       // Encoder fault from ZSW2_ENC
       "HMI_DB".Encoders."1BR".EncoderFault :=
       "DB_EncCom_1BR".EncoderFault;

       "HMI_DB".Encoders."1BR".ErrorCode :=
       "DB_EncCom_1BR".EncoderErrorCode;

       // Encoder alarm / warning from ZSW2_ENC
       "HMI_DB".Encoders."1BR".EncoderAlarm :=
       "DB_EncCom_1BR".EncoderAlarm;

       // Encoder sign-of-life is valid
       "HMI_DB".Encoders."1BR".EncoderLifeValid :=
       "DB_EncCom_1BR".EncoderLifeValid;


       // ============================================================
       // Preset status
       // ============================================================

       // Preset procedure is active
       "HMI_DB".Encoders."1BR".PresetBusy :=
       "DB_EncCom_1BR".PresetBusy;

       // Preset was done successfully
       "HMI_DB".Encoders."1BR".PresetDone :=
       "DB_EncCom_1BR".PresetDone;

       // Preset error
       "HMI_DB".Encoders."1BR".PresetError :=
       "DB_EncCom_1BR".PresetError;

       // Preset diagnostic status
       "HMI_DB".Encoders."1BR".PresetStatus :=
       "DB_EncCom_1BR".PresetStatus;


       // ============================================================
       // Telegram 89 diagnostic words
       // ============================================================

       // STW2_ENC: control word from PLC to encoder
       "HMI_DB".Encoders."1BR".STW2_ENC :=
       "DB_EncCom_1BR".PzdOutActual.STW2_ENC;

       // ZSW2_ENC: status word from encoder to PLC
       "HMI_DB".Encoders."1BR".ZSW2_ENC :=
       "DB_EncCom_1BR".PzdInActual.ZSW2_ENC;


       // ============================================================
       // General communication FB status
       // ============================================================

       // General diagnostic word of FB_Enc_Tlg89_Com
       "HMI_DB".Encoders."1BR".Status :=
       "DB_EncCom_1BR".Status;

       // -----------------------------------------------------------------------------
       // Масштабоване положення підйому 1BR.
       // -----------------------------------------------------------------------------

       "HMI_DB".Encoders."1BR".Position_mm :=
       LREAL_TO_REAL(
                     "DB_PosCorrection_1BR".ql_PositionCorrected_mm
       );

       "HMI_DB".Encoders."1BR".PositionRounded_mm :=
       "DB_PosCorrection_1BR".qd_PositionCorrectedRounded_mm;

       "HMI_DB".Encoders."1BR".PositionValid :=
       "DB_EncoderScaling".Enc_1BR.PositionValid;

       //======================================

   END_REGION

   //Енкодер пересування візка
   REGION Enc_3BR
       //*********************************
       //Енкодер пересування візка 3BR
       //*********************************

       // ============================================================
       // Main raw values
       // ============================================================

       // Raw position from encoder G1_XIST2
       "HMI_DB".Encoders."3BR".RawPosition :=
       "DB_EncCom_3BR".AbsolutePositionRaw;

       // Raw velocity from encoder NIST_B
       "HMI_DB".Encoders."3BR".RawVelocity :=
       "DB_EncCom_3BR".VelocityRaw;


       // ============================================================
       // Main encoder status
       // ============================================================

       // Encoder is ready for crane logic
       "HMI_DB".Encoders."3BR".EncoderReady :=
       "DB_EncCom_3BR".EncoderReady;

       // Raw position is valid
       "HMI_DB".Encoders."3BR".PositionDataValid :=
       "DB_EncCom_3BR".PositionDataValid;

       // Raw velocity is valid
       "HMI_DB".Encoders."3BR".VelocityDataValid :=
       "DB_EncCom_3BR".VelocityDataValid;

       // Communication fault or cyclic data fault
       "HMI_DB".Encoders."3BR".CommunicationFault :=
       "DB_EncCom_3BR".CommunicationFault;

       // Encoder fault from ZSW2_ENC
       "HMI_DB".Encoders."3BR".EncoderFault :=
       "DB_EncCom_3BR".EncoderFault;

       "HMI_DB".Encoders."3BR".ErrorCode :=
       "DB_EncCom_3BR".EncoderErrorCode;

       // Encoder alarm / warning from ZSW2_ENC
       "HMI_DB".Encoders."3BR".EncoderAlarm :=
       "DB_EncCom_3BR".EncoderAlarm;

       // Encoder sign-of-life is valid
       "HMI_DB".Encoders."3BR".EncoderLifeValid :=
       "DB_EncCom_3BR".EncoderLifeValid;


       // ============================================================
       // Preset status
       // ============================================================

       // Preset procedure is active
       "HMI_DB".Encoders."3BR".PresetBusy :=
       "DB_EncCom_3BR".PresetBusy;

       // Preset was done successfully
       "HMI_DB".Encoders."3BR".PresetDone :=
       "DB_EncCom_3BR".PresetDone;

       // Preset error
       "HMI_DB".Encoders."3BR".PresetError :=
       "DB_EncCom_3BR".PresetError;

       // Preset diagnostic status
       "HMI_DB".Encoders."3BR".PresetStatus :=
       "DB_EncCom_3BR".PresetStatus;


       // ============================================================
       // Telegram 89 diagnostic words
       // ============================================================

       // STW2_ENC: control word from PLC to encoder
       "HMI_DB".Encoders."3BR".STW2_ENC :=
       "DB_EncCom_3BR".PzdOutActual.STW2_ENC;

       // ZSW2_ENC: status word from encoder to PLC
       "HMI_DB".Encoders."3BR".ZSW2_ENC :=
       "DB_EncCom_3BR".PzdInActual.ZSW2_ENC;


       // ============================================================
       // General communication FB status
       // ============================================================

       // General diagnostic word of FB_Enc_Tlg89_Com
       "HMI_DB".Encoders."3BR".Status :=
       "DB_EncCom_3BR".Status;

       // -----------------------------------------------------------------------------
       // Масштабоване положення підйому 1BR.
       // -----------------------------------------------------------------------------

       "HMI_DB".Encoders."3BR".Position_mm :=
       LREAL_TO_REAL(
                     "DB_PosCorrection_3BR".ql_PositionCorrected_mm
       );

       "HMI_DB".Encoders."3BR".PositionRounded_mm :=
       "DB_PosCorrection_3BR".qd_PositionCorrectedRounded_mm;

       "HMI_DB".Encoders."3BR".PositionValid :=
       "DB_EncoderScaling".Enc_3BR.PositionValid;

       //======================================

   END_REGION

   //Енкодер#1 пересування крана
   REGION Enc_4BR1
       //*********************************
       //Енкодер пересування візка 3BR
       //*********************************

       // ============================================================
       // Main raw values
       // ============================================================

       // Raw position from encoder G1_XIST2
       "HMI_DB".Encoders."4BR1".RawPosition :=
       "DB_EncCom_4BR1".AbsolutePositionRaw;

       // Raw velocity from encoder NIST_B
       "HMI_DB".Encoders."4BR1".RawVelocity :=
       "DB_EncCom_4BR1".VelocityRaw;


       // ============================================================
       // Main encoder status
       // ============================================================

       // Encoder is ready for crane logic
       "HMI_DB".Encoders."4BR1".EncoderReady :=
       "DB_EncCom_4BR1".EncoderReady;

       // Raw position is valid
       "HMI_DB".Encoders."4BR1".PositionDataValid :=
       "DB_EncCom_4BR1".PositionDataValid;

       // Raw velocity is valid
       "HMI_DB".Encoders."4BR1".VelocityDataValid :=
       "DB_EncCom_4BR1".VelocityDataValid;

       // Communication fault or cyclic data fault
       "HMI_DB".Encoders."4BR1".CommunicationFault :=
       "DB_EncCom_4BR1".CommunicationFault;

       // Encoder fault from ZSW2_ENC
       "HMI_DB".Encoders."4BR1".EncoderFault :=
       "DB_EncCom_4BR1".EncoderFault;

       "HMI_DB".Encoders."4BR1".ErrorCode :=
       "DB_EncCom_4BR1".EncoderErrorCode;

       // Encoder alarm / warning from ZSW2_ENC
       "HMI_DB".Encoders."4BR1".EncoderAlarm :=
       "DB_EncCom_4BR1".EncoderAlarm;

       // Encoder sign-of-life is valid
       "HMI_DB".Encoders."4BR1".EncoderLifeValid :=
       "DB_EncCom_4BR1".EncoderLifeValid;


       // ============================================================
       // Preset status
       // ============================================================

       // Preset procedure is active
       "HMI_DB".Encoders."4BR1".PresetBusy :=
       "DB_EncCom_4BR1".PresetBusy;

       // Preset was done successfully
       "HMI_DB".Encoders."4BR1".PresetDone :=
       "DB_EncCom_4BR1".PresetDone;

       // Preset error
       "HMI_DB".Encoders."4BR1".PresetError :=
       "DB_EncCom_4BR1".PresetError;

       // Preset diagnostic status
       "HMI_DB".Encoders."4BR1".PresetStatus :=
       "DB_EncCom_4BR1".PresetStatus;


       // ============================================================
       // Telegram 89 diagnostic words
       // ============================================================

       // STW2_ENC: control word from PLC to encoder
       "HMI_DB".Encoders."4BR1".STW2_ENC :=
       "DB_EncCom_4BR1".PzdOutActual.STW2_ENC;

       // ZSW2_ENC: status word from encoder to PLC
       "HMI_DB".Encoders."4BR1".ZSW2_ENC :=
       "DB_EncCom_4BR1".PzdInActual.ZSW2_ENC;


       // ============================================================
       // General communication FB status
       // ============================================================

       // General diagnostic word of FB_Enc_Tlg89_Com
       "HMI_DB".Encoders."4BR1".Status :=
       "DB_EncCom_4BR1".Status;

       // -----------------------------------------------------------------------------
       // Масштабоване положення підйому 1BR.
       // -----------------------------------------------------------------------------

       "HMI_DB".Encoders."4BR1".Position_mm :=
       LREAL_TO_REAL(
                     "DB_PosCorrection_4BR1".ql_PositionCorrected_mm
       );

       "HMI_DB".Encoders."4BR1".PositionRounded_mm :=
       "DB_PosCorrection_4BR1".qd_PositionCorrectedRounded_mm;

       "HMI_DB".Encoders."4BR1".PositionValid :=
       "DB_EncoderScaling".Enc_4BR1.PositionValid;

       //======================================

   END_REGION

   //Енкодер#2 пересування крана
   REGION Enc_4BR2
       //*********************************
       //Енкодер пересування візка 3BR
       //*********************************

       // ============================================================
       // Main raw values
       // ============================================================

       // Raw position from encoder G1_XIST2
       "HMI_DB".Encoders."4BR2".RawPosition :=
       "DB_EncCom_4BR2".AbsolutePositionRaw;

       // Raw velocity from encoder NIST_B
       "HMI_DB".Encoders."4BR2".RawVelocity :=
       "DB_EncCom_4BR2".VelocityRaw;


       // ============================================================
       // Main encoder status
       // ============================================================

       // Encoder is ready for crane logic
       "HMI_DB".Encoders."4BR2".EncoderReady :=
       "DB_EncCom_4BR2".EncoderReady;

       // Raw position is valid
       "HMI_DB".Encoders."4BR2".PositionDataValid :=
       "DB_EncCom_4BR2".PositionDataValid;

       // Raw velocity is valid
       "HMI_DB".Encoders."4BR2".VelocityDataValid :=
       "DB_EncCom_4BR2".VelocityDataValid;

       // Communication fault or cyclic data fault
       "HMI_DB".Encoders."4BR2".CommunicationFault :=
       "DB_EncCom_4BR2".CommunicationFault;

       // Encoder fault from ZSW2_ENC
       "HMI_DB".Encoders."4BR2".EncoderFault :=
       "DB_EncCom_4BR2".EncoderFault;

       "HMI_DB".Encoders."4BR2".ErrorCode :=
       "DB_EncCom_4BR2".EncoderErrorCode;

       // Encoder alarm / warning from ZSW2_ENC
       "HMI_DB".Encoders."4BR2".EncoderAlarm :=
       "DB_EncCom_4BR2".EncoderAlarm;

       // Encoder sign-of-life is valid
       "HMI_DB".Encoders."4BR2".EncoderLifeValid :=
       "DB_EncCom_4BR2".EncoderLifeValid;


       // ============================================================
       // Preset status
       // ============================================================

       // Preset procedure is active
       "HMI_DB".Encoders."4BR2".PresetBusy :=
       "DB_EncCom_4BR2".PresetBusy;

       // Preset was done successfully
       "HMI_DB".Encoders."4BR2".PresetDone :=
       "DB_EncCom_4BR2".PresetDone;

       // Preset error
       "HMI_DB".Encoders."4BR2".PresetError :=
       "DB_EncCom_4BR2".PresetError;

       // Preset diagnostic status
       "HMI_DB".Encoders."4BR2".PresetStatus :=
       "DB_EncCom_4BR2".PresetStatus;


       // ============================================================
       // Telegram 89 diagnostic words
       // ============================================================

       // STW2_ENC: control word from PLC to encoder
       "HMI_DB".Encoders."4BR2".STW2_ENC :=
       "DB_EncCom_4BR2".PzdOutActual.STW2_ENC;

       // ZSW2_ENC: status word from encoder to PLC
       "HMI_DB".Encoders."4BR2".ZSW2_ENC :=
       "DB_EncCom_4BR2".PzdInActual.ZSW2_ENC;


       // ============================================================
       // General communication FB status
       // ============================================================

       // General diagnostic word of FB_Enc_Tlg89_Com
       "HMI_DB".Encoders."4BR2".Status :=
       "DB_EncCom_4BR2".Status;

       // -----------------------------------------------------------------------------
       // Масштабоване положення підйому 1BR.
       // -----------------------------------------------------------------------------

       "HMI_DB".Encoders."4BR2".Position_mm :=
       LREAL_TO_REAL(
                     "DB_PosCorrection_4BR2".ql_PositionCorrected_mm
       );

       "HMI_DB".Encoders."4BR2".PositionRounded_mm :=
       "DB_PosCorrection_4BR2".qd_PositionCorrectedRounded_mm;

       "HMI_DB".Encoders."4BR2".PositionValid :=
       "DB_EncoderScaling".Enc_4BR2.PositionValid;

       //======================================

   END_REGION
END_FUNCTION

FUNCTION "FC_EncoderScale" : Void   // FC82, LAD
{ S7_Optimized_Access := 'TRUE' }
VERSION : 0.1
   VAR_INPUT
      Enable : Bool;   // Загальний дозвіл роботи функції.
      RawPosition : DInt;   // Поточне сире абсолютне положення енкодера.
      RawPositionValid : Bool;   // TRUE — поточне raw-положення достовірне.
      RawPoint1 : DInt;   // Сире значення енкодера у першій контрольній точці.
      PositionPoint1_mm : LReal;   // Координата першої контрольної точки, мм.
      RawPoint2 : DInt;   // Сире значення енкодера у другій контрольній точці.
      PositionPoint2_mm : LReal;   // Координата другої контрольної точки, мм.
   END_VAR
   VAR_OUTPUT
      Position_mm : LReal;   // Розраховане положення механізму, мм.
      PositionRounded_mm : DInt;   // Положення, округлене до цілого міліметра.
      PositionValid : Bool;   // Розраховане положення достовірне. / Результат достовірний і знаходиться в налаштованому діапазоні.
      CalculationValid : Bool;   // Математичний розрахунок виконано за достовірним raw-сигналом.
      ConfigurationValid : Bool;   // Контрольні точки задані коректно.
      InConfiguredRange : Bool;   // Поточне raw-значення знаходиться між двома контрольними точками масштабування. / Поточне raw-значення знаходиться між RawPoint1 і RawPoint2.
      BelowConfiguredRange : Bool;   // Raw-значення нижче мінімальної контрольної raw-точки.
      AboveConfiguredRange : Bool;   // Raw-значення вище максимальної контрольної raw-точки.
      Scale_mm_per_count : LReal;   // Розрахований коефіцієнт масштабування.
      Status : Word;   // Діагностичне слово функції.
   END_VAR
   VAR_TEMP
      RawSpan : LReal;   // Різниця між двома raw-точками.
      PositionSpan_mm : LReal;   // Різниця координат між двома точками, мм.
      RawDelta : LReal;   // Відхилення поточного raw від першої точки.
      RawMinimum : DInt;   // Менша із двох raw-точок.
      RawMaximum : DInt;   // Більша із двох raw-точок.
      CalculatedPosition_mm : LReal;   // Тимчасовий результат масштабування.
   END_VAR
BEGIN

REGION Network 2 (SCL): Розраховане положення механізму, мм.
   // ============================================================
   // 1. Початкові значення виходів
   // ============================================================

   #Position_mm := 0.0;
   #PositionRounded_mm := DINT#0;

   #PositionValid := FALSE;
   #CalculationValid := FALSE;
   #ConfigurationValid := FALSE;

   #InConfiguredRange := FALSE;
   #BelowConfiguredRange := FALSE;
   #AboveConfiguredRange := FALSE;

   #Scale_mm_per_count := 0.0;
   #Status := W#16#0000;

   #RawSpan := 0.0;
   #PositionSpan_mm := 0.0;
   #RawDelta := 0.0;

   #RawMinimum := DINT#0;
   #RawMaximum := DINT#0;

   #CalculatedPosition_mm := 0.0;


   // ============================================================
   // 2. Перевірка дозволу роботи
   // ============================================================

   IF NOT #Enable THEN

       // Bit 0: функція вимкнена.
       #Status := #Status OR W#16#0001;

       RETURN;

   END_IF;


   // ============================================================
   // 3. Перевірка конфігурації контрольних точок
   // ============================================================

   IF #RawPoint1 = #RawPoint2 THEN

       // Bit 2: однакові raw-точки.
       #Status := #Status OR W#16#0004;

   END_IF;


   IF #PositionPoint1_mm = #PositionPoint2_mm THEN

       // Bit 3: однакові координати контрольних точок.
       #Status := #Status OR W#16#0008;

   END_IF;


   #ConfigurationValid :=
   (#RawPoint1 <> #RawPoint2)
   AND
   (#PositionPoint1_mm <> #PositionPoint2_mm);


   IF NOT #ConfigurationValid THEN
       RETURN;
   END_IF;


   // ============================================================
   // 4. Визначення мінімальної та максимальної raw-точок
   // ============================================================

   IF #RawPoint1 < #RawPoint2 THEN

       #RawMinimum := #RawPoint1;
       #RawMaximum := #RawPoint2;

   ELSE

       #RawMinimum := #RawPoint2;
       #RawMaximum := #RawPoint1;

   END_IF;


   // ============================================================
   // 5. Перевірка знаходження raw у налаштованому діапазоні
   // ============================================================

   #BelowConfiguredRange :=
   #RawPosition < #RawMinimum;

   #AboveConfiguredRange :=
   #RawPosition > #RawMaximum;

   #InConfiguredRange :=
   NOT #BelowConfiguredRange
   AND NOT #AboveConfiguredRange;


   IF NOT #InConfiguredRange THEN

       // Bit 4: raw-положення поза налаштованим діапазоном.
       #Status := #Status OR W#16#0010;

   END_IF;


   IF #BelowConfiguredRange THEN

       // Bit 7: raw нижче налаштованого діапазону.
       #Status := #Status OR W#16#0080;

   END_IF;


   IF #AboveConfiguredRange THEN

       // Bit 8: raw вище налаштованого діапазону.
       #Status := #Status OR W#16#0100;

   END_IF;


   // ============================================================
   // 6. Розрахунок коефіцієнта масштабування
   // ============================================================

   // Перетворення виконується до віднімання,
   // щоб уникнути переповнення типу DINT.
   #RawSpan :=
   DINT_TO_LREAL(#RawPoint2)
   - DINT_TO_LREAL(#RawPoint1);

   #PositionSpan_mm :=
   #PositionPoint2_mm
   - #PositionPoint1_mm;

   #Scale_mm_per_count :=
   #PositionSpan_mm
   / #RawSpan;


   // ============================================================
   // 7. Перевірка достовірності вхідного raw-положення
   // ============================================================

   IF NOT #RawPositionValid THEN

       // Bit 1: вхідне raw-положення недостовірне.
       #Status := #Status OR W#16#0002;

       RETURN;

   END_IF;


   // ============================================================
   // 8. Масштабування raw-положення у міліметри
   // ============================================================

   #RawDelta :=
   DINT_TO_LREAL(#RawPosition)
   - DINT_TO_LREAL(#RawPoint1);

   #CalculatedPosition_mm :=
   #PositionPoint1_mm
   + (#RawDelta * #Scale_mm_per_count);

   #Position_mm :=
   #CalculatedPosition_mm;

   #PositionRounded_mm :=
   LREAL_TO_DINT(#CalculatedPosition_mm);

   #CalculationValid := TRUE;

   // Bit 5: математичний розрахунок виконано.
   #Status := #Status OR W#16#0020;


   // ============================================================
   // 9. Формування остаточної валідності положення
   // ============================================================

   #PositionValid :=
   #ConfigurationValid
   AND #RawPositionValid;

   IF #PositionValid THEN

       // Bit 6: результат придатний для штатного використання.
       #Status := #Status OR W#16#0040;

   END_IF;
END_REGION
END_FUNCTION

FUNCTION "FC_AxisProgramLimits" : Void   // FC83, LAD
{ S7_Optimized_Access := 'TRUE' }
VERSION : 0.1
   VAR_INPUT
      Enable : Bool;   // Загальний дозвіл роботи
      Position_mm : LReal;   // Поточне масштабоване положення
      PositionValid : Bool;   // TRUE = положення достовірне
      ProgStopNegative_mm : LReal;   // Нижня програмна межа
      ProgStopPositive_mm : LReal;   // Верхня програмна межа
   END_VAR
   VAR_OUTPUT
      ProgStopNegative : Bool;   // TRUE = досягнута нижня програмна межа
      ProgStopPositive : Bool;   // TRUE = досягнута верхня програмна межа
      ConfigurationValid : Bool;   // TRUE = межі задані коректно
   END_VAR
BEGIN

REGION Network 2 (SCL): Програмні межі
   #ProgStopNegative := FALSE;
   #ProgStopPositive := FALSE;

   #ConfigurationValid :=
   #ProgStopNegative_mm < #ProgStopPositive_mm;

   IF #Enable
       AND #PositionValid
       AND #ConfigurationValid THEN

       #ProgStopNegative :=
       #Position_mm <= #ProgStopNegative_mm;

       #ProgStopPositive :=
       #Position_mm >= #ProgStopPositive_mm;

   END_IF;
END_REGION
END_FUNCTION

FUNCTION "FC_TrolleyPositionLimits" : Void   // FC84, SCL
{ S7_Optimized_Access := 'TRUE' }
VERSION : 0.1
   VAR_INPUT
      Enable : Bool;   // Загальний дозвіл роботи функції
      Position_mm : LReal;   // Поточне скориговане положення механізму візка, мм
      PositionValid : Bool;   // TRUE = положення енкодера достовірне
      BackBuffer_mm : LReal;   // Крайня механічна позиція / буфер назад
      BackEmergencyLimit_mm : LReal;   // Позиція аварійного апаратного кінцевика назад
      BackEncoderLimit_mm : LReal;   // Програмна межа по енкодеру назад
      BackPreStop_mm : LReal;   // Технологічний передзупин назад
      ForwardPreStop_mm : LReal;   // Технологічний передзупин вперед
      ForwardEncoderLimit_mm : LReal;   // Програмна межа по енкодеру вперед
      ForwardEmergencyLimit_mm : LReal;   // Позиція аварійного апаратного кінцевика вперед
      ForwardBuffer_mm : LReal;   // Крайня механічна позиція / буфер вперед
      VirtualOffset_mm : LReal;   // Віртуальне зміщення системи координат, мм
   END_VAR
   VAR_OUTPUT
      BackBuffer : Bool;   // TRUE = досягнута або перевищена позиція буфера назад
      BackEmergencyLimit : Bool;   // TRUE = досягнута позиція аварійного кінцевика назад
      BackEncoderLimit : Bool;   // TRUE = досягнута програмна межа по енкодеру назад
      BackPreStop : Bool;   // TRUE = візок знаходиться в зоні технологічного передзупину назад
      ForwardPreStop : Bool;   // TRUE = візок знаходиться в зоні технологічного передзупину вперед
      ForwardEncoderLimit : Bool;   // TRUE = досягнута програмна межа по енкодеру вперед
      ForwardEmergencyLimit : Bool;   // TRUE = досягнута позиція аварійного кінцевика вперед
      ForwardBuffer : Bool;   // TRUE = досягнута або перевищена позиція буфера вперед
      ConfigurationValid : Bool;   // TRUE = усі координатні уставки задані у правильній послідовності
   END_VAR
BEGIN
   // ============================================================
   // FC_TrolleyPositionLimits
   // Контроль координатних меж і зон механізму візка
   //
   // Негативний напрямок = назад
   // Позитивний напрямок = вперед
   //
   // Послідовність координат:
   //
   // Назад:
   // Буфер -> Аварійний кінцевик -> Межа по енкодеру -> Передзупин
   //
   // Вперед:
   // Передзупин -> Межа по енкодеру -> Аварійний кінцевик -> Буфер
   // ============================================================


   // ============================================================
   // 1. Початкові значення виходів
   // ============================================================

   #BackBuffer := FALSE;
   #BackEmergencyLimit := FALSE;
   #BackEncoderLimit := FALSE;
   #BackPreStop := FALSE;

   #ForwardPreStop := FALSE;
   #ForwardEncoderLimit := FALSE;
   #ForwardEmergencyLimit := FALSE;
   #ForwardBuffer := FALSE;


   // ============================================================
   // 2. Перевірка конфігурації
   //
   // Усі координатні межі повинні бути задані послідовно
   // від заднього буфера до переднього буфера.
   // ============================================================

   #ConfigurationValid :=
   (#BackBuffer_mm < #BackEmergencyLimit_mm)
   AND (#BackEmergencyLimit_mm < #BackEncoderLimit_mm)
   AND (#BackEncoderLimit_mm < #BackPreStop_mm)
   AND (#BackPreStop_mm < #ForwardPreStop_mm)
   AND (#ForwardPreStop_mm < #ForwardEncoderLimit_mm)
   AND (#ForwardEncoderLimit_mm < #ForwardEmergencyLimit_mm)
   AND (#ForwardEmergencyLimit_mm < #ForwardBuffer_mm);


   // ============================================================
   // 3. Розрахунок координатних меж
   //
   // Контроль виконується тільки за умов:
   // - функція дозволена;
   // - положення енкодера достовірне;
   // - конфігурація координатних меж коректна.
   // ============================================================

   IF #Enable
       AND #PositionValid
       AND #ConfigurationValid
   THEN

       // ========================================================
       // 3.1 Рух назад
       //
       // При русі назад координата візка зменшується.
       // Вихід стає TRUE після досягнення відповідної межі.
       // ========================================================

       // Досягнута зона технологічного передзупину назад.
       #BackPreStop :=
       #Position_mm <= (#BackPreStop_mm + #VirtualOffset_mm);

       // Досягнута програмна межа по енкодеру назад.
       #BackEncoderLimit :=
       #Position_mm <= (#BackEncoderLimit_mm + #VirtualOffset_mm);

       // Досягнута позиція аварійного апаратного кінцевика назад.
       #BackEmergencyLimit :=
       #Position_mm <= (#BackEmergencyLimit_mm + #VirtualOffset_mm);

       // Досягнута крайня механічна позиція / буфер назад.
       #BackBuffer :=
       #Position_mm <= (#BackBuffer_mm + #VirtualOffset_mm);


       // ========================================================
       // 3.2 Рух вперед
       //
       // При русі вперед координата візка збільшується.
       // Вихід стає TRUE після досягнення відповідної межі.
       // ========================================================

       // Досягнута зона технологічного передзупину вперед.
       #ForwardPreStop :=
       #Position_mm >= (#ForwardPreStop_mm + #VirtualOffset_mm);

       // Досягнута програмна межа по енкодеру вперед.
       #ForwardEncoderLimit :=
       #Position_mm >=(#ForwardEncoderLimit_mm + #VirtualOffset_mm);

       // Досягнута позиція аварійного апаратного кінцевика вперед.
       #ForwardEmergencyLimit :=
       #Position_mm >= (#ForwardEmergencyLimit_mm + #VirtualOffset_mm);

       // Досягнута крайня механічна позиція / буфер вперед.
       #ForwardBuffer :=
       #Position_mm >= (#ForwardBuffer_mm + #VirtualOffset_mm);

   END_IF;
END_FUNCTION

FUNCTION "FC_HoistPositionLimits" : Void   // FC85, SCL
{ S7_Optimized_Access := 'TRUE' }
VERSION : 0.1
   VAR_INPUT
      Enable : Bool;   // Загальний дозвіл роботи функції
      Position_mm : LReal;   // Поточне скориговане положення механізму підйому, мм
      PositionValid : Bool;   // TRUE = положення енкодера достовірне
      DownEndPosition_mm : LReal;   // Крайня нижня позиція механізму
      DownEmergencyLimit_mm : LReal;   // Позиція аварійного кінцевика при опусканні
      DownEncoderLimit_mm : LReal;   // Програмна межа по енкодеру при опусканні
      DownPreStop_mm : LReal;   // Технологічний передзупин при опусканні
      UpPreStop_mm : LReal;   // Технологічний передзупин при підйомі
      UpEncoderLimit_mm : LReal;   // Програмна межа по енкодеру при підйомі
      UpEmergencyLimit_mm : LReal;   // Позиція аварійного кінцевика при підйомі
      UpEndPosition_mm : LReal;   // Крайня верхня позиція механізму
      VirtualOffset_mm : LReal;   // Віртуальне зміщення системи координат, мм
   END_VAR
   VAR_OUTPUT
      DownEndPosition : Bool;   // Досягнута крайня нижня позиція
      DownEmergencyLimit : Bool;   // Досягнута позиція аварійного кінцевика при опусканні
      DownEncoderLimit : Bool;   // Досягнута програмна межа по енкодеру при опусканні
      DownPreStop : Bool;   // Активна зона технологічного передзупину при опусканні
      UpPreStop : Bool;   // Активна зона технологічного передзупину при підйомі
      UpEncoderLimit : Bool;   // Досягнута програмна межа по енкодеру при підйомі
      UpEmergencyLimit : Bool;   // Досягнута позиція аварійного кінцевика при підйомі
      UpEndPosition : Bool;   // Досягнута крайня верхня позиція
      ConfigurationValid : Bool;   // TRUE = координатні межі задані коректно
   END_VAR
BEGIN
   // ============================================================
   // FC_HoistPositionLimits
   // Контроль координатних меж механізму підйому
   //
   // Підйом     = позитивний напрямок руху.
   // Опускання  = негативний напрямок руху.
   //
   // При підйомі координата збільшується.
   // При опусканні координата зменшується.
   //
   // Послідовність меж при опусканні:
   // Низ -> Аварійний кінцевик -> Межа по енкодеру -> Передзупин
   //
   // Послідовність меж при підйомі:
   // Передзупин -> Межа по енкодеру -> Аварійний кінцевик -> Верх
   // ============================================================


   // ============================================================
   // 1. Початкові значення виходів
   // ============================================================

   #DownEndPosition := FALSE;
   #DownEmergencyLimit := FALSE;
   #DownEncoderLimit := FALSE;
   #DownPreStop := FALSE;

   #UpPreStop := FALSE;
   #UpEncoderLimit := FALSE;
   #UpEmergencyLimit := FALSE;
   #UpEndPosition := FALSE;


   // ============================================================
   // 2. Перевірка конфігурації
   //
   // Координатні межі повинні послідовно збільшуватись
   // від крайньої нижньої позиції до крайньої верхньої позиції.
   // ============================================================

   #ConfigurationValid :=
   (#DownEndPosition_mm < #DownEmergencyLimit_mm)
   AND (#DownEmergencyLimit_mm < #DownEncoderLimit_mm)
   AND (#DownEncoderLimit_mm < #DownPreStop_mm)
   AND (#DownPreStop_mm < #UpPreStop_mm)
   AND (#UpPreStop_mm < #UpEncoderLimit_mm)
   AND (#UpEncoderLimit_mm < #UpEmergencyLimit_mm)
   AND (#UpEmergencyLimit_mm < #UpEndPosition_mm);


   // ============================================================
   // 3. Розрахунок координатних меж
   //
   // Контроль виконується тільки за умов:
   // - функція дозволена;
   // - положення енкодера достовірне;
   // - конфігурація координатних меж коректна.
   // ============================================================

   IF #Enable
       AND #PositionValid
       AND #ConfigurationValid
   THEN

       // ========================================================
       // 3.1 Опускання
       //
       // Опускання є негативним напрямком руху.
       // При опусканні координата зменшується.
       // ========================================================

       // Досягнута зона технологічного передзупину при опусканні.
       #DownPreStop :=
       #Position_mm <= (#DownPreStop_mm + #VirtualOffset_mm);

       // Досягнута програмна межа по енкодеру при опусканні.
       #DownEncoderLimit :=
       #Position_mm <= (#DownEncoderLimit_mm + #VirtualOffset_mm);

       // Досягнута позиція аварійного апаратного кінцевика
       // при опусканні.
       #DownEmergencyLimit :=
       #Position_mm <= (#DownEmergencyLimit_mm + #VirtualOffset_mm);

       // Досягнута крайня нижня позиція механізму.
       #DownEndPosition :=
       #Position_mm <= (#DownEndPosition_mm + #VirtualOffset_mm);


       // ========================================================
       // 3.2 Підйом
       //
       // Підйом є позитивним напрямком руху.
       // При підйомі координата збільшується.
       // ========================================================

       // Досягнута зона технологічного передзупину при підйомі.
       #UpPreStop :=
       #Position_mm >= (#UpPreStop_mm + #VirtualOffset_mm);

       // Досягнута програмна межа по енкодеру при підйомі.
       #UpEncoderLimit :=
       #Position_mm >= (#UpEncoderLimit_mm + #VirtualOffset_mm);

       // Досягнута позиція аварійного апаратного кінцевика
       // при підйомі.
       #UpEmergencyLimit :=
       #Position_mm >= (#UpEmergencyLimit_mm + #VirtualOffset_mm);

       // Досягнута крайня верхня позиція механізму.
       #UpEndPosition :=
       #Position_mm >= (#UpEndPosition_mm + #VirtualOffset_mm);

   END_IF;
END_FUNCTION

FUNCTION "FC_BridgePositionLimits" : Void   // FC86, SCL
{ S7_Optimized_Access := 'TRUE' }
VERSION : 0.1
   VAR_INPUT
      Enable : Bool;   // Загальний дозвіл роботи функції
      Position_mm : LReal;   // Поточне скориговане положення механізму моста, мм
      PositionValid : Bool;   // TRUE = положення енкодера достовірне
      LeftBuffer_mm : LReal;   // Позиція буфера зліва
      LeftEmergencyLimit_mm : LReal;   // Позиція аварійного кінцевика зліва
      LeftEncoderLimit_mm : LReal;   // Програмна межа по енкодеру зліва
      LeftPreStop_mm : LReal;   // Технологічний передзупин при русі вліво
      LeftZoneLimit_mm : LReal;   // Ліва координатна межа зони
      RightZoneLimit_mm : LReal;   // Права координатна межа зони
      RightPreStop_mm : LReal;   // Технологічний передзупин при русі вправо
      RightEncoderLimit_mm : LReal;   // Програмна межа по енкодеру справа
      RightEmergencyLimit_mm : LReal;   // Позиція аварійного кінцевика справа
      RightBuffer_mm : LReal;   // Позиція буфера справа
      VirtualOffset_mm : LReal;   // Віртуальне зміщення системи координат, мм
   END_VAR
   VAR_OUTPUT
      LeftBuffer : Bool;   // Досягнута позиція буфера зліва
      LeftEmergencyLimit : Bool;   // Досягнута позиція аварійного кінцевика зліва
      LeftEncoderLimit : Bool;   // Досягнута програмна межа по енкодеру зліва
      LeftPreStop : Bool;   // Досягнута технологічна межа при русі вліво
      LeftZoneLimit : Bool;   // Досягнута ліва межа зони
      RightZoneLimit : Bool;   // Досягнута права межа зони
      RightPreStop : Bool;   // Досягнута технологічна межа при русі вправо
      RightEncoderLimit : Bool;   // Досягнута програмна межа по енкодеру справа
      RightEmergencyLimit : Bool;   // Досягнута позиція аварійного кінцевика справа
      RightBuffer : Bool;   // Досягнута позиція буфера справа
      ConfigurationValid : Bool;   // TRUE = координатні межі задані коректно
   END_VAR
BEGIN
   // ============================================================
   // FC_BridgePositionLimits
   // Контроль координатних меж механізму моста крана
   //
   // Вправо = позитивний напрямок руху.
   // Вліво  = негативний напрямок руху.
   //
   // При русі вправо координата збільшується.
   // При русі вліво координата зменшується.
   //
   // Послідовність координат:
   //
   // Вліво:
   // Буфер -> Аварійний кінцевик -> Межа по енкодеру
   // -> Технологічний передзупин -> Ліва межа зони
   //
   // Вправо:
   // Права межа зони -> Технологічний передзупин
   // -> Межа по енкодеру -> Аварійний кінцевик -> Буфер
   // ============================================================


   // ============================================================
   // 1. Початкові значення виходів
   // ============================================================

   #LeftBuffer := FALSE;
   #LeftEmergencyLimit := FALSE;
   #LeftEncoderLimit := FALSE;
   #LeftPreStop := FALSE;
   #LeftZoneLimit := FALSE;

   #RightZoneLimit := FALSE;
   #RightPreStop := FALSE;
   #RightEncoderLimit := FALSE;
   #RightEmergencyLimit := FALSE;
   #RightBuffer := FALSE;


   // ============================================================
   // 2. Перевірка конфігурації
   //
   // Координатні межі повинні послідовно збільшуватись
   // від лівого буфера до правого буфера.
   // ============================================================

   #ConfigurationValid :=
   (#LeftBuffer_mm < #LeftEmergencyLimit_mm)
   AND (#LeftEmergencyLimit_mm < #LeftEncoderLimit_mm)
   AND (#LeftEncoderLimit_mm < #LeftPreStop_mm)
   AND (#LeftPreStop_mm < #LeftZoneLimit_mm)
   AND (#LeftZoneLimit_mm < #RightZoneLimit_mm)
   AND (#RightZoneLimit_mm < #RightPreStop_mm)
   AND (#RightPreStop_mm < #RightEncoderLimit_mm)
   AND (#RightEncoderLimit_mm < #RightEmergencyLimit_mm)
   AND (#RightEmergencyLimit_mm < #RightBuffer_mm);


   // ============================================================
   // 3. Розрахунок координатних меж
   //
   // Контроль виконується тільки за умов:
   // - функція дозволена;
   // - положення енкодера достовірне;
   // - конфігурація координатних меж коректна.
   // ============================================================

   IF #Enable
       AND #PositionValid
       AND #ConfigurationValid
   THEN

       // ========================================================
       // 3.1 Рух вліво
       //
       // Вліво є негативним напрямком руху.
       // При русі вліво координата зменшується.
       // ========================================================

       // Досягнута ліва координатна межа зони.
       #LeftZoneLimit :=
       #Position_mm <= (#LeftZoneLimit_mm + #VirtualOffset_mm);

       // Досягнута зона технологічного передзупину
       // при русі вліво.
       #LeftPreStop :=
       #Position_mm <= (#LeftPreStop_mm + #VirtualOffset_mm);

       // Досягнута програмна межа по енкодеру зліва.
       #LeftEncoderLimit :=
       #Position_mm <= (#LeftEncoderLimit_mm + #VirtualOffset_mm);

       // Досягнута позиція аварійного апаратного кінцевика
       // зліва.
       #LeftEmergencyLimit :=
       #Position_mm <= (#LeftEmergencyLimit_mm + #VirtualOffset_mm);

       // Досягнута позиція буфера зліва.
       #LeftBuffer :=
       #Position_mm <= (#LeftBuffer_mm + #VirtualOffset_mm);


       // ========================================================
       // 3.2 Рух вправо
       //
       // Вправо є позитивним напрямком руху.
       // При русі вправо координата збільшується.
       // ========================================================

       // Досягнута права координатна межа зони.
       #RightZoneLimit :=
       #Position_mm >= (#RightZoneLimit_mm + #VirtualOffset_mm);

       // Досягнута зона технологічного передзупину
       // при русі вправо.
       #RightPreStop :=
       #Position_mm >= (#RightPreStop_mm + #VirtualOffset_mm);

       // Досягнута програмна межа по енкодеру справа.
       #RightEncoderLimit :=
       #Position_mm >= (#RightEncoderLimit_mm + #VirtualOffset_mm);

       // Досягнута позиція аварійного апаратного кінцевика
       // справа.
       #RightEmergencyLimit :=
       #Position_mm >= (#RightEmergencyLimit_mm + #VirtualOffset_mm);

       // Досягнута позиція буфера справа.
       #RightBuffer :=
       #Position_mm >= (#RightBuffer_mm + #VirtualOffset_mm);

   END_IF;
END_FUNCTION

// ===== library types =====

TYPE "AnCfg"
   STRUCT
      VRaw : Int;   // Raw value (from input channel)
      LORaw : Int;   // Raw value LO limit
      HIRaw : Int;   // RAW value HI limit
      Val : Real;   // Output value
      LOEng : Real;   // Engineering (scaled) minimum value
      HIEng : Real;   // Engineering (scaled) maximum value
      FVal : Real;   // Filtered value
      PhyVal : Real;   // Physical value (mA)
      LOSP : Real;   // LO setpoint
      LOLOSP : Real;   // LO-LO setpoint
      HISP : Real;   // HI setpoint
      HIHISP : Real;   // HI-HI setpoint
      Hyst : Real;   // Hysteresis in real units
      SimVal : Real;   // Value for simulation
      LOEn : Bool;   // LO warning enabled
      LOLOEn : Bool;   // LO-LO Alarm enabled
      HIEn : Bool;   // HI warning enabled
      HIHIEn : Bool;   // HI-HI Alarm enabled
      LO : Bool;   // Low level is reached
      LOLO : Bool;   // Low Low level is reached
      HI : Bool;   // High level is reached
      HIHI : Bool;   // High High level is reached
      SML : Bool;   // Output value is simulated
      Reset : Bool;   // Reset
      STS : Int;   // Status
      T_FLTR : Int;   // Filtering time, x0.01 seconds
      Text : WString;   // Tag name
      Chanal : WString;   // Chanal
   END_STRUCT;
END_TYPE

(* ===== HMI "HMI_RT_1" =====
system functions are stored by id; their names below are inferred from use
connection "HMI_Connection_1": ETHERNET, S7_1500_OMS

HMI tags "Default tag table"
   "Tag_ScreenNumber" : UInt, internal
   "xAllwaysFalse" : Bool, internal
   "iStep" : Int, internal

HMI tags "DI"
   "HMI_DB_IO_Tags_InCnf_DigIn_0_0" : DigICfg = PLC HMI_DB.IO_Tags.InCnf.DigIn_0_0, 1 s
   "HMI_DB_IO_Tags_InCnf_DigIn_0_1" : DigICfg = PLC HMI_DB.IO_Tags.InCnf.DigIn_0_1 AT %DB1.DBW0, 1 s
   "HMI_DB_IO_Tags_InCnf_DigIn_0_2" : DigICfg = PLC HMI_DB.IO_Tags.InCnf.DigIn_0_2 AT %DB1.DBW0, 1 s
   "HMI_DB_IO_Tags_InCnf_DigIn_0_3" : DigICfg = PLC HMI_DB.IO_Tags.InCnf.DigIn_0_3 AT %DB1.DBW0, 1 s
   "HMI_DB_IO_Tags_InCnf_DigIn_0_4" : DigICfg = PLC HMI_DB.IO_Tags.InCnf.DigIn_0_4 AT %DB1.DBW0, 1 s
   "HMI_DB_IO_Tags_InCnf_DigIn_0_5" : DigICfg = PLC HMI_DB.IO_Tags.InCnf.DigIn_0_5 AT %DB1.DBW0, 1 s
   "HMI_DB_IO_Tags_InCnf_DigIn_0_6" : DigICfg = PLC HMI_DB.IO_Tags.InCnf.DigIn_0_6 AT %DB1.DBW0, 1 s
   "HMI_DB_IO_Tags_InCnf_DigIn_0_7" : DigICfg = PLC HMI_DB.IO_Tags.InCnf.DigIn_0_7 AT %DB1.DBW0, 1 s
   "HMI_DB_IO_Tags_InCnf_DigIn_1_0" : DigICfg = PLC HMI_DB.IO_Tags.InCnf.DigIn_1_0 AT %DB1.DBW0, 1 s
   "HMI_DB_IO_Tags_InCnf_DigIn_1_1" : DigICfg = PLC HMI_DB.IO_Tags.InCnf.DigIn_1_1 AT %DB1.DBW0, 1 s
   "HMI_DB_IO_Tags_InCnf_DigIn_1_2" : DigICfg = PLC HMI_DB.IO_Tags.InCnf.DigIn_1_2 AT %DB1.DBW0, 1 s
   "HMI_DB_IO_Tags_InCnf_DigIn_1_3" : DigICfg = PLC HMI_DB.IO_Tags.InCnf.DigIn_1_3 AT %DB1.DBW0, 1 s
   "HMI_DB_IO_Tags_InCnf_DigIn_1_4" : DigICfg = PLC HMI_DB.IO_Tags.InCnf.DigIn_1_4 AT %DB1.DBW0, 1 s
   "HMI_DB_IO_Tags_InCnf_DigIn_1_5" : DigICfg = PLC HMI_DB.IO_Tags.InCnf.DigIn_1_5 AT %DB1.DBW0, 1 s
   "HMI_DB_IO_Tags_InCnf_DigIn_1_6" : DigICfg = PLC HMI_DB.IO_Tags.InCnf.DigIn_1_6 AT %DB1.DBW0, 1 s
   "HMI_DB_IO_Tags_InCnf_DigIn_1_7" : DigICfg = PLC HMI_DB.IO_Tags.InCnf.DigIn_1_7 AT %DB1.DBW0, 1 s
   "HMI_DB_IO_Tags_InCnf_DigIn_2_0" : DigICfg = PLC HMI_DB.IO_Tags.InCnf.DigIn_2_0 AT %DB1.DBW0, 1 s
   "HMI_DB_IO_Tags_InCnf_DigIn_2_1" : DigICfg = PLC HMI_DB.IO_Tags.InCnf.DigIn_2_1 AT %DB1.DBW0, 1 s
   "HMI_DB_IO_Tags_InCnf_DigIn_2_2" : DigICfg = PLC HMI_DB.IO_Tags.InCnf.DigIn_2_2 AT %DB1.DBW0, 1 s
   "HMI_DB_IO_Tags_InCnf_DigIn_2_3" : DigICfg = PLC HMI_DB.IO_Tags.InCnf.DigIn_2_3 AT %DB1.DBW0, 1 s
   "HMI_DB_IO_Tags_InCnf_DigIn_2_4" : DigICfg = PLC HMI_DB.IO_Tags.InCnf.DigIn_2_4 AT %DB1.DBW0, 1 s
   "HMI_DB_IO_Tags_InCnf_DigIn_2_5" : DigICfg = PLC HMI_DB.IO_Tags.InCnf.DigIn_2_5 AT %DB1.DBW0, 1 s
   "HMI_DB_IO_Tags_InCnf_DigIn_2_6" : DigICfg = PLC HMI_DB.IO_Tags.InCnf.DigIn_2_6 AT %DB1.DBW0, 1 s
   "HMI_DB_IO_Tags_InCnf_DigIn_2_7" : DigICfg = PLC HMI_DB.IO_Tags.InCnf.DigIn_2_7 AT %DB1.DBW0, 1 s
   "HMI_DB_IO_Tags_InCnf_DigIn_3_0" : DigICfg = PLC HMI_DB.IO_Tags.InCnf.DigIn_3_0 AT %DB1.DBW0, 1 s
   "HMI_DB_IO_Tags_InCnf_DigIn_3_1" : DigICfg = PLC HMI_DB.IO_Tags.InCnf.DigIn_3_1 AT %DB1.DBW0, 1 s
   "HMI_DB_IO_Tags_InCnf_DigIn_3_2" : DigICfg = PLC HMI_DB.IO_Tags.InCnf.DigIn_3_2 AT %DB1.DBW0, 1 s
   "HMI_DB_IO_Tags_InCnf_DigIn_3_3" : DigICfg = PLC HMI_DB.IO_Tags.InCnf.DigIn_3_3 AT %DB1.DBW0, 1 s
   "HMI_DB_IO_Tags_InCnf_DigIn_3_4" : DigICfg = PLC HMI_DB.IO_Tags.InCnf.DigIn_3_4 AT %DB1.DBW0, 1 s
   "HMI_DB_IO_Tags_InCnf_DigIn_3_5" : DigICfg = PLC HMI_DB.IO_Tags.InCnf.DigIn_3_5 AT %DB1.DBW0, 1 s
   "HMI_DB_IO_Tags_InCnf_DigIn_3_6" : DigICfg = PLC HMI_DB.IO_Tags.InCnf.DigIn_3_6 AT %DB1.DBW0, 1 s
   "HMI_DB_IO_Tags_InCnf_DigIn_3_7" : DigICfg = PLC HMI_DB.IO_Tags.InCnf.DigIn_3_7 AT %DB1.DBW0, 1 s
   "HMI_DB_IO_Tags_InCnf_DigIn_4_0" : DigICfg = PLC HMI_DB.IO_Tags.InCnf.DigIn_4_0 AT %DB1.DBW0, 1 s
   "HMI_DB_IO_Tags_InCnf_DigIn_4_1" : DigICfg = PLC HMI_DB.IO_Tags.InCnf.DigIn_4_1 AT %DB1.DBW0, 1 s
   "HMI_DB_IO_Tags_InCnf_DigIn_4_2" : DigICfg = PLC HMI_DB.IO_Tags.InCnf.DigIn_4_2 AT %DB1.DBW0, 1 s
   "HMI_DB_IO_Tags_InCnf_DigIn_4_3" : DigICfg = PLC HMI_DB.IO_Tags.InCnf.DigIn_4_3 AT %DB1.DBW0, 1 s
   "HMI_DB_IO_Tags_InCnf_DigIn_4_4" : DigICfg = PLC HMI_DB.IO_Tags.InCnf.DigIn_4_4 AT %DB1.DBW0, 1 s
   "HMI_DB_IO_Tags_InCnf_DigIn_4_5" : DigICfg = PLC HMI_DB.IO_Tags.InCnf.DigIn_4_5 AT %DB1.DBW0, 1 s
   "HMI_DB_IO_Tags_InCnf_DigIn_4_6" : DigICfg = PLC HMI_DB.IO_Tags.InCnf.DigIn_4_6 AT %DB1.DBW0, 1 s
   "HMI_DB_IO_Tags_InCnf_DigIn_4_7" : DigICfg = PLC HMI_DB.IO_Tags.InCnf.DigIn_4_7 AT %DB1.DBW0, 1 s
   "HMI_DB_IO_Tags_InCnf_DigIn_5_0" : DigICfg = PLC HMI_DB.IO_Tags.InCnf.DigIn_5_0 AT %DB1.DBW0, 1 s
   "HMI_DB_IO_Tags_InCnf_DigIn_5_1" : DigICfg = PLC HMI_DB.IO_Tags.InCnf.DigIn_5_1 AT %DB1.DBW0, 1 s
   "HMI_DB_IO_Tags_InCnf_DigIn_5_2" : DigICfg = PLC HMI_DB.IO_Tags.InCnf.DigIn_5_2 AT %DB1.DBW0, 1 s
   "HMI_DB_IO_Tags_InCnf_DigIn_5_3" : DigICfg = PLC HMI_DB.IO_Tags.InCnf.DigIn_5_3 AT %DB1.DBW0, 1 s
   "HMI_DB_IO_Tags_InCnf_DigIn_5_4" : DigICfg = PLC HMI_DB.IO_Tags.InCnf.DigIn_5_4 AT %DB1.DBW0, 1 s
   "HMI_DB_IO_Tags_InCnf_DigIn_5_5" : DigICfg = PLC HMI_DB.IO_Tags.InCnf.DigIn_5_5 AT %DB1.DBW0, 1 s
   "HMI_DB_IO_Tags_InCnf_DigIn_5_6" : DigICfg = PLC HMI_DB.IO_Tags.InCnf.DigIn_5_6 AT %DB1.DBW0, 1 s
   "HMI_DB_IO_Tags_InCnf_DigIn_5_7" : DigICfg = PLC HMI_DB.IO_Tags.InCnf.DigIn_5_7 AT %DB1.DBW0, 1 s
   "HMI_DB_IO_Tags_InCnf_DigIn_6_0" : DigICfg = PLC HMI_DB.IO_Tags.InCnf.DigIn_6_0 AT %DB1.DBW0, 1 s
   "HMI_DB_IO_Tags_InCnf_DigIn_6_1" : DigICfg = PLC HMI_DB.IO_Tags.InCnf.DigIn_6_1 AT %DB1.DBW0, 1 s
   "HMI_DB_IO_Tags_InCnf_DigIn_6_2" : DigICfg = PLC HMI_DB.IO_Tags.InCnf.DigIn_6_2 AT %DB1.DBW0, 1 s
   "HMI_DB_IO_Tags_InCnf_DigIn_6_3" : DigICfg = PLC HMI_DB.IO_Tags.InCnf.DigIn_6_3 AT %DB1.DBW0, 1 s
   "HMI_DB_IO_Tags_InCnf_DigIn_6_4" : DigICfg = PLC HMI_DB.IO_Tags.InCnf.DigIn_6_4 AT %DB1.DBW0, 1 s
   "HMI_DB_IO_Tags_InCnf_DigIn_6_5" : DigICfg = PLC HMI_DB.IO_Tags.InCnf.DigIn_6_5 AT %DB1.DBW0, 1 s
   "HMI_DB_IO_Tags_InCnf_DigIn_6_6" : DigICfg = PLC HMI_DB.IO_Tags.InCnf.DigIn_6_6 AT %DB1.DBW0, 1 s
   "HMI_DB_IO_Tags_InCnf_DigIn_6_7" : DigICfg = PLC HMI_DB.IO_Tags.InCnf.DigIn_6_7 AT %DB1.DBW0, 1 s
   "HMI_DB_IO_Tags_InCnf_DigIn_7_0" : DigICfg = PLC HMI_DB.IO_Tags.InCnf.DigIn_7_0 AT %DB1.DBW0, 1 s
   "HMI_DB_IO_Tags_InCnf_DigIn_7_1" : DigICfg = PLC HMI_DB.IO_Tags.InCnf.DigIn_7_1 AT %DB1.DBW0, 1 s
   "HMI_DB_IO_Tags_InCnf_DigIn_7_2" : DigICfg = PLC HMI_DB.IO_Tags.InCnf.DigIn_7_2 AT %DB1.DBW0, 1 s
   "HMI_DB_IO_Tags_InCnf_DigIn_7_3" : DigICfg = PLC HMI_DB.IO_Tags.InCnf.DigIn_7_3 AT %DB1.DBW0, 1 s
   "HMI_DB_IO_Tags_InCnf_DigIn_7_4" : DigICfg = PLC HMI_DB.IO_Tags.InCnf.DigIn_7_4 AT %DB1.DBW0, 1 s
   "HMI_DB_IO_Tags_InCnf_DigIn_7_5" : DigICfg = PLC HMI_DB.IO_Tags.InCnf.DigIn_7_5 AT %DB1.DBW0, 1 s
   "HMI_DB_IO_Tags_InCnf_DigIn_7_6" : DigICfg = PLC HMI_DB.IO_Tags.InCnf.DigIn_7_6 AT %DB1.DBW0, 1 s
   "HMI_DB_IO_Tags_InCnf_DigIn_7_7" : DigICfg = PLC HMI_DB.IO_Tags.InCnf.DigIn_7_7 AT %DB1.DBW0, 1 s

HMI tags "Internaltags"
   "iVisibilityA1.2" : Bool, internal
   "iVisibilityA1.3" : Bool, internal
   "iVisibilityDevices" : Int, internal

HMI tags "DO"
   "HMI_DB_IO_Tags_OutCfg_DigOut_0_0" : DigOCfg = PLC HMI_DB.IO_Tags.OutCfg.DigOut_0_0, 1 s
   "HMI_DB_IO_Tags_OutCfg_DigOut_0_1" : DigOCfg = PLC HMI_DB.IO_Tags.OutCfg.DigOut_0_1, 1 s
   "HMI_DB_IO_Tags_OutCfg_DigOut_0_2" : DigOCfg = PLC HMI_DB.IO_Tags.OutCfg.DigOut_0_2, 1 s
   "HMI_DB_IO_Tags_OutCfg_DigOut_0_3" : DigOCfg = PLC HMI_DB.IO_Tags.OutCfg.DigOut_0_3, 1 s
   "HMI_DB_IO_Tags_OutCfg_DigOut_0_4" : DigOCfg = PLC HMI_DB.IO_Tags.OutCfg.DigOut_0_4, 1 s
   "HMI_DB_IO_Tags_OutCfg_DigOut_0_5" : DigOCfg = PLC HMI_DB.IO_Tags.OutCfg.DigOut_0_5, 1 s
   "HMI_DB_IO_Tags_OutCfg_DigOut_0_6" : DigOCfg = PLC HMI_DB.IO_Tags.OutCfg.DigOut_0_6, 1 s
   "HMI_DB_IO_Tags_OutCfg_DigOut_0_7" : DigOCfg = PLC HMI_DB.IO_Tags.OutCfg.DigOut_0_7, 1 s
   "HMI_DB_IO_Tags_OutCfg_DigOut_1_0" : DigOCfg = PLC HMI_DB.IO_Tags.OutCfg.DigOut_1_0, 1 s
   "HMI_DB_IO_Tags_OutCfg_DigOut_1_1" : DigOCfg = PLC HMI_DB.IO_Tags.OutCfg.DigOut_1_1, 1 s
   "HMI_DB_IO_Tags_OutCfg_DigOut_1_2" : DigOCfg = PLC HMI_DB.IO_Tags.OutCfg.DigOut_1_2, 1 s
   "HMI_DB_IO_Tags_OutCfg_DigOut_1_3" : DigOCfg = PLC HMI_DB.IO_Tags.OutCfg.DigOut_1_3, 1 s
   "HMI_DB_IO_Tags_OutCfg_DigOut_1_4" : DigOCfg = PLC HMI_DB.IO_Tags.OutCfg.DigOut_1_4, 1 s
   "HMI_DB_IO_Tags_OutCfg_DigOut_1_5" : DigOCfg = PLC HMI_DB.IO_Tags.OutCfg.DigOut_1_5, 1 s
   "HMI_DB_IO_Tags_OutCfg_DigOut_1_6" : DigOCfg = PLC HMI_DB.IO_Tags.OutCfg.DigOut_1_6, 1 s
   "HMI_DB_IO_Tags_OutCfg_DigOut_1_7" : DigOCfg = PLC HMI_DB.IO_Tags.OutCfg.DigOut_1_7, 1 s

HMI tags "AI"
   "HMI_DB_IO_Tags_InAnCfg_AnIn_0" : AnICfg = PLC HMI_DB.IO_Tags.InAnCfg.AnIn_0, 1 s
   "HMI_DB_IO_Tags_InAnCfg_AnIn_1" : AnICfg = PLC HMI_DB.IO_Tags.InAnCfg.AnIn_1, 1 s
   "HMI_DB_IO_Tags_InAnCfg_AnIn_2" : AnICfg = PLC HMI_DB.IO_Tags.InAnCfg.AnIn_2, 1 s
   "HMI_DB_IO_Tags_InAnCfg_AnIn_3" : AnICfg = PLC HMI_DB.IO_Tags.InAnCfg.AnIn_3, 1 s
   "HMI_DB_IO_Tags_InAnCfg_AnIn_4" : AnICfg = PLC HMI_DB.IO_Tags.InAnCfg.AnIn_4, 1 s
   "HMI_DB_IO_Tags_InAnCfg_AnIn_5" : AnICfg = PLC HMI_DB.IO_Tags.InAnCfg.AnIn_5, 1 s
   "HMI_DB_IO_Tags_InAnCfg_AnIn_6" : AnICfg = PLC HMI_DB.IO_Tags.InAnCfg.AnIn_6, 1 s
   "HMI_DB_IO_Tags_InAnCfg_AnIn_7" : AnICfg = PLC HMI_DB.IO_Tags.InAnCfg.AnIn_7, 1 s

HMI tags "Encoders"
   "HMI_DB_Encoders_1BR" : UDT_HMI_Encoder_View = PLC HMI_DB.Encoders.1BR, 1 s
   "HMI_DB_Encoders_3BR" : UDT_HMI_Encoder_View = PLC HMI_DB.Encoders.3BR AT %DB1.DBW0, 1 s
   "HMI_DB_Encoders_4BR1" : UDT_HMI_Encoder_View = PLC HMI_DB.Encoders.4BR1 AT %DB1.DBW0, 1 s
   "HMI_DB_Encoders_4BR2" : UDT_HMI_Encoder_View = PLC HMI_DB.Encoders.4BR2 AT %DB1.DBW0, 1 s

HMI tags "PSMErrors"
   "HMI_DB_Alarms_Contactor_AlarmWord1" : Word = PLC HMI_DB.Alarms.Contactor.AlarmWord1 AT %DB1.DBW0, 1 s
   "HMI_DB_Alarms_Contactor_AlarmWord2" : Word = PLC HMI_DB.Alarms.Contactor.AlarmWord2 AT %DB1.DBW0, 1 s
   "HMI_DB_Alarms_Contactor_AlarmWord3" : Word = PLC HMI_DB.Alarms.Contactor.AlarmWord3 AT %DB1.DBW0, 1 s
   "HMI_DB_PSM_LC_Alarm" : Bool = PLC HMI_DB.PSM.LC_Alarm AT %DB1.DBW0, 1 s

HMI tags "PSM"
   "HMI_DB_PSM_Line_contactor_On" : Bool = PLC HMI_DB.PSM.Line_contactor_On, 1 s
   "HMI_DB_PSM_Control_contactor_220V_On" : Bool = PLC HMI_DB.PSM.Control_contactor_220V_On, 1 s
   "HMI_DB_PSM_Input_voltage_control_380V_On" : Bool = PLC HMI_DB.PSM.Input_voltage_control_380V_On, 1 s
   "HMI_DB_PSM_Heating_circuit_breaker_220V_On" : Bool = PLC HMI_DB.PSM.Heating_circuit_breaker_220V_On, 1 s
   "HMI_DB_PSM_Brake_protection_On" : Bool = PLC HMI_DB.PSM.Brake_protection_On, 1 s
   "HMI_DB_PSM_Transformer_6T1_380V_On" : Bool = PLC HMI_DB.PSM.Transformer_6T1_380V_On, 1 s
   "HMI_DB_PSM_Transformer_sec_circuit_breaker_6T1_380V_On" : Bool = PLC HMI_DB.PSM.Transformer_sec_circuit_breaker_6T1_380V_On, 1 s
   "HMI_DB_PSM_Power_switch_6KV_380V_On" : Bool = PLC HMI_DB.PSM.Power_switch_6KV_380V_On, 1 s
   "HMI_DB_PSM_ID_Control_circuit_breaker_220V_On" : Bool = PLC HMI_DB.PSM.ID_Control_circuit_breaker_220V_On, 1 s
   "HMI_DB_PSM_ID_ORP_power_circuit_breaker_220V_On" : Bool = PLC HMI_DB.PSM.ID_ORP_power_circuit_breaker_220V_On, 1 s
   "HMI_DB_PSM_ID_Line_contactor_from_remote_control_On" : Bool = PLC HMI_DB.PSM.ID_Line_contactor_from_remote_control_On, 1 s
   "HMI_DB_PSM_Transformer_9T1_380V_On" : Bool = PLC HMI_DB.PSM.Transformer_9T1_380V_On, 1 s
   "HMI_DB_PSM_Repair_lighting_switch_12V_On" : Bool = PLC HMI_DB.PSM.Repair_lighting_switch_12V_On, 1 s
   "HMI_DB_PSM_Cabinet_circuit_breaker_220V_On" : Bool = PLC HMI_DB.PSM.Cabinet_circuit_breaker_220V_On, 1 s
   "HMI_DB_PSM_CMD_Line_contactor_enable_permission" : Bool = PLC HMI_DB.PSM.CMD_Line_contactor_enable_permission, 1 s
   "HMI_DB_PSM_CMD_Line_contactor_Off" : Bool = PLC HMI_DB.PSM.CMD_Line_contactor_Off, 1 s
   "HMI_DB_PSM_HL_Line_contactor_On" : Bool = PLC HMI_DB.Messages.Crane.wMessageWord1, 1 s
   "HMI_DB_PSM_HL_Input_voltage_abnormal" : Bool = PLC HMI_DB.PSM.HL_Input_voltage_abnormal, 1 s
   "HMI_DB_PSM_Zero_Protection" : Bool = PLC HMI_DB.PSM.Zero_Protection AT %DB1.DBX0.0, 1 s
   "Data_base_Profinet_Ok" : Bool = PLC HMI_DB.Diagnostics.Profinet_Ok AT %DB1.DBX0.0, 1 s
   "HMI_DB_PSM_ColumnEnable" : Bool = PLC HMI_DB.PSM.ColumnEnable AT %DB1.DBX0.0, 1 s
   "HMI_DB_FireAlarm_Active" : Bool = PLC HMI_DB.FireAlarm.Active AT %DB1.DBX0.0, 1 s

HMI tags "Sensors"
   "HMI_DB_Sensors_Cabinet_heating_control_SU1" : Bool = PLC HMI_DB.Sensors.Cabinet_heating_control_SU1, 1 s
   "HMI_DB_Sensors_Seismic_sensor" : Bool = PLC HMI_DB.Sensors.Seismic_sensor, 1 s
   "HMI_DB_Sensors_Drum_rotation_control" : Bool = PLC HMI_DB.Sensors.Drum_rotation_control, 1 s
   "HMI_DB_Sensors_CMD_Bell_On" : Bool = PLC HMI_DB.Sensors.CMD_Bell_On, 500 ms

HMI tags "RemoteControl"
   "HMI_DB_Remote_control" : udtRemCtrl = PLC HMI_DB.Remote_control, 1 s
   "HMI_DB_Remote_control_1" : Bool = PLC HMI_DB.Remote_control.Btn_Bell AT %DB1.DBX0.0, 1 s

HMI tags "LiftingMechanism"
   "HMI_DB_Lifting_mechanism_Work_control" : Bool = PLC HMI_DB.Lifting_mechanism.Work_control, 1 s
   "HMI_DB_Lifting_mechanism_Brake_wear_control" : Bool = PLC HMI_DB.Lifting_mechanism.Brake_wear_control, 1 s
   "HMI_DB_Lifting_mechanism_MD_disconnected_from_drive" : Bool = PLC HMI_DB.Lifting_mechanism.MD_disconnected_from_drive, 1 s
   "HMI_DB_Lifting_mechanism_Thermal_protection_braking_resistor" : Bool = PLC HMI_DB.Lifting_mechanism.Thermal_protection_braking_resistor, 1 s
   "HMI_DB_Lifting_mechanism_NSP_Upward_movement" : Bool = PLC HMI_DB.Lifting_mechanism.NSP_Upward_movement, 1 s
   "HMI_DB_Lifting_mechanism_NSP_Downward_movement" : Bool = PLC HMI_DB.Lifting_mechanism.NSP_Downward_movement, 1 s
   "HMI_DB_Lifting_mechanism_WP_Upward_movement" : Bool = PLC HMI_DB.Lifting_mechanism.WP_Upward_movement, 1 s
   "HMI_DB_Lifting_mechanism_WP_Downward_movement" : Bool = PLC HMI_DB.Lifting_mechanism.WP_Downward_movement, 1 s
   "HMI_DB_Lifting_mechanism_Exceeding_rated_load_115%" : Bool = PLC HMI_DB.Lifting_mechanism.Exceeding_rated_load_115%, 1 s
   "HMI_DB_Lifting_mechanism_Loosening_ropes" : Bool = PLC HMI_DB.Lifting_mechanism.Loosening_ropes, 1 s
   "HMI_DB_Lifting_mechanism_Motor_temperature_protection" : Bool = PLC HMI_DB.Lifting_mechanism.Motor_temperature_protection, 1 s
   "HMI_DB_Lifting_mechanism_1YB1_Brake released" : Bool = PLC HMI_DB.Lifting_mechanism."1YB1_Brake released", 1 s
   "HMI_DB_Lifting_mechanism_1YB1_Brake_applied" : Bool = PLC HMI_DB.Lifting_mechanism.1YB1_Brake_applied, 1 s
   "HMI_DB_Lifting_mechanism_1YB1_Thickness_brake_pads_normal" : Bool = PLC HMI_DB.Lifting_mechanism.1YB1_Thickness_brake_pads_normal, 1 s
   "HMI_DB_Lifting_mechanism_1YB2_Brake released" : Bool = PLC HMI_DB.Lifting_mechanism."1YB2_Brake released", 1 s
   "HMI_DB_Lifting_mechanism_1YB2_Brake_applied" : Bool = PLC HMI_DB.Lifting_mechanism.1YB2_Brake_applied, 1 s
   "HMI_DB_Lifting_mechanism_1YB2_WP_MPP_disconnected_from_brake" : Bool = PLC HMI_DB.Lifting_mechanism.1YB2_WP_MPP_disconnected_from_brake, 1 s
   "HMI_DB_Lifting_mechanism_1YB1_Brake_rectifier_protection" : Bool = PLC HMI_DB.Lifting_mechanism.1YB1_Brake_rectifier_protection, 1 s
   "HMI_DB_Lifting_mechanism_1YB2_Brake_rectifier_protection" : Bool = PLC HMI_DB.Lifting_mechanism.1YB2_Brake_rectifier_protection, 1 s
   "HMI_DB_Lifting_mechanism_CMD_Service_brake_On" : Bool = PLC HMI_DB.Lifting_mechanism.CMD_Service_brake_On, 1 s
   "HMI_DB_Lifting_mechanism_CMD_Built-in_brake_On" : Bool = PLC HMI_DB.Lifting_mechanism.CMD_Built-in_brake_On, 1 s
   "HMI_DB_Lifting_mechanism_CMD_Emergency_brake_On" : Bool = PLC HMI_DB.Lifting_mechanism.CMD_Emergency_brake_On, 1 s
   "HMI_DB_Lifting_mechanism_HL_Drive_ready" : Bool = PLC HMI_DB.Lifting_mechanism.HL_Drive_ready, 1 s
   "HMI_DB_Lifting_mechanism_Torque_control" : Real = PLC HMI_DB.Lifting_mechanism.Torque_control, 1 s
   "HMI_DB_Lifting_mechanism_LM_Alarm" : Bool = PLC HMI_DB.Lifting_mechanism.LM_Alarm AT %DB1.DBX0.0, 1 s
   "HMI_DB_Lifting_mechanism_LM_Status" : Word = PLC HMI_DB.Lifting_mechanism.LM_Status AT %DB1.DBX0.0, 1 s
   "HMI_DB_Lifting_mechanism_NSP_Enable_movement" : Bool = PLC HMI_DB.Lifting_mechanism.NSP_Enable_movement AT %DB1.DBX0.0, 1 s
   "HMI_DB_Lifting_mechanism_SecondSpeedUp" : Bool = PLC HMI_DB.Lifting_mechanism.SecondSpeedUp AT %DB1.DBX0.0, 1 s
   "HMI_DB_Lifting_mechanism_SecondSpeedDown" : Bool = PLC HMI_DB.Lifting_mechanism.SecondSpeedDown, 1 s
   "HMI_DB_Lifting_mechanism_FirstSpeedUp" : Bool = PLC HMI_DB.Lifting_mechanism.FirstSpeedUp AT %DB1.DBX0.0, 1 s
   "HMI_DB_Lifting_mechanism_FirstSpeedDown" : Bool = PLC HMI_DB.Lifting_mechanism.FirstSpeedDown AT %DB1.DBX0.0, 1 s
   "HMI_DB_Calibration_Hoist_Active" : Bool = PLC HMI_DB.Calibration.Hoist.Active AT %DB1.DBX0.0, 1 s
   "HMI_DB_Calibration_Hoist_Calibrated" : Bool = PLC HMI_DB.Calibration.Hoist.Calibrated AT %DB1.DBX0.0, 1 s
   "HMI_DB_Calibration_Hoist_Fault" : Bool = PLC HMI_DB.Calibration.Hoist.Fault AT %DB1.DBX0.0, 1 s
   "HMI_DB_Calibration_Hoist_Aborted" : Bool = PLC HMI_DB.Calibration.Hoist.Aborted AT %DB1.DBX0.0, 1 s
   "HMI_DB_Calibration_Hoist_CurrentStep" : UInt = PLC HMI_DB.Calibration.Hoist.CurrentStep AT %DB1.DBX0.0, 1 s
   "HMI_DB_Calibration_Hoist_CompletedSteps" : DWord = PLC HMI_DB.Calibration.Hoist.CompletedSteps AT %DB1.DBX0.0, 1 s
   "HMI_DB_Calibration_Hoist_Reference1K1" : Bool = PLC HMI_DB.Calibration.Hoist.Reference1K1 AT %DB1.DBX0.0, 1 s
   "HMI_DB_Calibration_Hoist_Position_mm" : DInt = PLC HMI_DB.Calibration.Hoist.Position_mm AT %DB1.DBX0.0, 1 s
   "HMI_DB_Calibration_Hoist_DriveVelocity_rpm" : Real = PLC HMI_DB.Calibration.Hoist.DriveVelocity_rpm AT %DB1.DBX0.0, 1 s
   "HMI_DB_Calibration_Hoist_TimerRemaining" : Time = PLC HMI_DB.Calibration.Hoist.TimerRemaining AT %DB1.DBX0.0, 1 s
   "HMI_DB_Calibration_Hoist_Steps_Completed_Step10" : Bool = PLC HMI_DB.Calibration.Hoist.Steps_Completed.Step10 AT %DB1.DBX0.0, 1 s
   "HMI_DB_Calibration_Hoist_Steps_Completed_Step20" : Bool = PLC HMI_DB.Calibration.Hoist.Steps_Completed.Step20 AT %DB1.DBX0.0, 1 s
   "HMI_DB_Calibration_Hoist_Steps_Completed_Step30" : Bool = PLC HMI_DB.Calibration.Hoist.Steps_Completed.Step30 AT %DB1.DBX0.0, 1 s
   "HMI_DB_Calibration_Hoist_Steps_Completed_Step40" : Bool = PLC HMI_DB.Calibration.Hoist.Steps_Completed.Step40 AT %DB1.DBX0.0, 1 s
   "HMI_DB_Calibration_Hoist_Steps_Completed_Step50" : Bool = PLC HMI_DB.Calibration.Hoist.Steps_Completed.Step50 AT %DB1.DBX0.0, 1 s
   "HMI_DB_Calibration_Hoist_Steps_Completed_Step60" : Bool = PLC HMI_DB.Calibration.Hoist.Steps_Completed.Step60 AT %DB1.DBX0.0, 1 s
   "HMI_DB_Calibration_Hoist_Steps_Completed_Step70" : Bool = PLC HMI_DB.Calibration.Hoist.Steps_Completed.Step70 AT %DB1.DBX0.0, 1 s
   "HMI_DB_Calibration_Hoist_Steps_Completed_Step80" : Bool = PLC HMI_DB.Calibration.Hoist.Steps_Completed.Step80 AT %DB1.DBX0.0, 1 s
   "HMI_DB_Calibration_Hoist_Steps_Completed_Step90" : Bool = PLC HMI_DB.Calibration.Hoist.Steps_Completed.Step90 AT %DB1.DBX0.0, 1 s
   "HMI_DB_Calibration_Hoist_Steps_Completed_Step100" : Bool = PLC HMI_DB.Calibration.Hoist.Steps_Completed.Step100 AT %DB1.DBX0.0, 1 s
   "HMI_DB_Calibration_Hoist_Steps_Completed_Step110" : Bool = PLC HMI_DB.Calibration.Hoist.Steps_Completed.Step110 AT %DB1.DBX0.0, 1 s
   "HMI_DB_Calibration_Hoist_Steps_Completed_Step120" : Bool = PLC HMI_DB.Calibration.Hoist.Steps_Completed.Step120 AT %DB1.DBX0.0, 1 s
   "HMI_DB_Calibration_Hoist_Steps_Completed_Step130" : Bool = PLC HMI_DB.Calibration.Hoist.Steps_Completed.Step130 AT %DB1.DBX0.0, 1 s
   "HMI_DB_Calibration_Hoist_Steps_Active_Step10" : Bool = PLC HMI_DB.Calibration.Hoist.Steps_Active.Step10 AT %DB1.DBX0.0, 1 s
   "HMI_DB_Calibration_Hoist_Steps_Active_Step20" : Bool = PLC HMI_DB.Calibration.Hoist.Steps_Active.Step20 AT %DB1.DBX0.0, 1 s
   "HMI_DB_Calibration_Hoist_Steps_Active_Step30" : Bool = PLC HMI_DB.Calibration.Hoist.Steps_Active.Step30 AT %DB1.DBX0.0, 1 s
   "HMI_DB_Calibration_Hoist_Steps_Active_Step40" : Bool = PLC HMI_DB.Calibration.Hoist.Steps_Active.Step40 AT %DB1.DBX0.0, 1 s
   "HMI_DB_Calibration_Hoist_Steps_Active_Step50" : Bool = PLC HMI_DB.Calibration.Hoist.Steps_Active.Step50 AT %DB1.DBX0.0, 1 s
   "HMI_DB_Calibration_Hoist_Steps_Active_Step60" : Bool = PLC HMI_DB.Calibration.Hoist.Steps_Active.Step60 AT %DB1.DBX0.0, 1 s
   "HMI_DB_Calibration_Hoist_Steps_Active_Step70" : Bool = PLC HMI_DB.Calibration.Hoist.Steps_Active.Step70 AT %DB1.DBX0.0, 1 s
   "HMI_DB_Calibration_Hoist_Steps_Active_Step80" : Bool = PLC HMI_DB.Calibration.Hoist.Steps_Active.Step80 AT %DB1.DBX0.0, 1 s
   "HMI_DB_Calibration_Hoist_Steps_Active_Step90" : Bool = PLC HMI_DB.Calibration.Hoist.Steps_Active.Step90 AT %DB1.DBX0.0, 1 s
   "HMI_DB_Calibration_Hoist_Steps_Active_Step100" : Bool = PLC HMI_DB.Calibration.Hoist.Steps_Active.Step100 AT %DB1.DBX0.0, 1 s
   "HMI_DB_Calibration_Hoist_Steps_Active_Step110" : Bool = PLC HMI_DB.Calibration.Hoist.Steps_Active.Step110 AT %DB1.DBX0.0, 1 s
   "HMI_DB_Calibration_Hoist_Steps_Active_Step120" : Bool = PLC HMI_DB.Calibration.Hoist.Steps_Active.Step120 AT %DB1.DBX0.0, 1 s
   "HMI_DB_Calibration_Hoist_Steps_Active_Step130" : Bool = PLC HMI_DB.Calibration.Hoist.Steps_Active.Step130 AT %DB1.DBX0.0, 1 s
   "HMI_DB_Calibration_Hoist_TimerRemaining_Min" : UInt = PLC HMI_DB.Calibration.Hoist.TimerRemaining_Min AT %DB1.DBX0.0, 1 s
   "HMI_DB_Calibration_Hoist_TimerRemaining_Sec" : UInt = PLC HMI_DB.Calibration.Hoist.TimerRemaining_Sec AT %DB1.DBX0.0, 1 s
   "HMI_DB_Calibration_Hoist_Diagnostics_EncoderControlHealthy" : Bool = PLC HMI_DB.Calibration.Hoist.Diagnostics.EncoderControlHealthy AT %DB1.DBX0.0, 1 s
   "HMI_DB_Calibration_Hoist_Diagnostics_StartupDataConsistent" : Bool = PLC HMI_DB.Calibration.Hoist.Diagnostics.StartupDataConsistent AT %DB1.DBX0.0, 1 s
   "HMI_DB_Calibration_Hoist_Diagnostics_NoMovementWithoutCommand" : Bool = PLC HMI_DB.Calibration.Hoist.Diagnostics.NoMovementWithoutCommand AT %DB1.DBX0.0, 1 s
   "HMI_DB_Calibration_Hoist_Diagnostics_NoManualMovementDetected" : Bool = PLC HMI_DB.Calibration.Hoist.Diagnostics.NoManualMovementDetected AT %DB1.DBX0.0, 1 s
   "HMI_DB_Calibration_Hoist_Diagnostics_EncoderUpdatesDuringMotion" : Bool = PLC HMI_DB.Calibration.Hoist.Diagnostics.EncoderUpdatesDuringMotion AT %DB1.DBX0.0, 1 s
   "HMI_DB_Calibration_Hoist_Diagnostics_EncoderReplacementNotDetected" : Bool = PLC HMI_DB.Calibration.Hoist.Diagnostics.EncoderReplacementNotDetected AT %DB1.DBX0.0, 1 s

HMI tags "TrolleyMovementMechanism"
   "HMI_DB_Trolley_movement_mechanism_Engine_temperature_protection" : Bool = PLC HMI_DB.Trolley_movement_mechanism.Engine_temperature_protection, 1 s
   "HMI_DB_Trolley_movement_mechanism_NSP_Forward_movement" : Bool = PLC HMI_DB.Trolley_movement_mechanism.NSP_Forward_movement, 1 s
   "HMI_DB_Trolley_movement_mechanism_WP_Forward_movement" : Bool = PLC HMI_DB.Trolley_movement_mechanism.WP_Forward_movement, 1 s
   "HMI_DB_Trolley_movement_mechanism_NSP_Backward_movement" : Bool = PLC HMI_DB.Trolley_movement_mechanism.NSP_Backward_movement, 1 s
   "HMI_DB_Trolley_movement_mechanism_WP_Backward_movement" : Bool = PLC HMI_DB.Trolley_movement_mechanism.WP_Backward_movement, 1 s
   "HMI_DB_Trolley_movement_mechanism_MD_disconnected_from_drive" : Bool = PLC HMI_DB.Trolley_movement_mechanism.MD_disconnected_from_drive, 1 s
   "HMI_DB_Trolley_movement_mechanism_Motor_temperature_protection" : Bool = PLC HMI_DB.Trolley_movement_mechanism.Motor_temperature_protection, 1 s
   "HMI_DB_Trolley_movement_mechanism_CMD_Service_brake_On" : Bool = PLC HMI_DB.Trolley_movement_mechanism.CMD_Service_brake_On, 1 s
   "HMI_DB_Trolley_movement_mechanism_HL_Drive_ready" : Bool = PLC HMI_DB.Trolley_movement_mechanism.HL_Drive_ready, 1 s
   "HMI_DB_Trolley_movement_mechanism_TM_Status" : Word = PLC HMI_DB.Trolley_movement_mechanism.TM_Status AT %DB1.DBX0.0, 1 s
   "HMI_DB_Trolley_movement_mechanism_NSP_Enable_movement" : Bool = PLC HMI_DB.Trolley_movement_mechanism.NSP_Enable_movement AT %DB1.DBX0.0, 1 s
   "HMI_DB_Trolley_movement_mechanism_SecondSpeedForwrd" : Bool = PLC HMI_DB.Trolley_movement_mechanism.SecondSpeedForward AT %DB1.DBX0.0, 1 s
   "HMI_DB_Trolley_movement_mechanism_SecondSpeedBackward" : Bool = PLC HMI_DB.Trolley_movement_mechanism.SecondSpeedBackward AT %DB1.DBX0.0, 1 s
   "HMI_DB_Trolley_movement_mechanism_FirstSpeedForward" : Bool = PLC HMI_DB.Trolley_movement_mechanism.FirstSpeedForward AT %DB1.DBX0.0, 1 s
   "HMI_DB_Trolley_movement_mechanism_FirstSpeedBackward" : Bool = PLC HMI_DB.Trolley_movement_mechanism.FirstSpeedBackward AT %DB1.DBX0.0, 1 s
   "HMI_DB_Calibration_Trolley_Active" : Bool = PLC HMI_DB.Calibration.Trolley.Active AT %DB1.DBX0.0, 1 s
   "HMI_DB_Calibration_Trolley_Calibrated" : Bool = PLC HMI_DB.Calibration.Trolley.Calibrated AT %DB1.DBX0.0, 1 s
   "HMI_DB_Calibration_Trolley_Fault" : Bool = PLC HMI_DB.Calibration.Trolley.Fault AT %DB1.DBX0.0, 1 s
   "HMI_DB_Calibration_Trolley_Aborted" : Bool = PLC HMI_DB.Calibration.Trolley.Aborted AT %DB1.DBX0.0, 1 s
   "HMI_DB_Calibration_Trolley_HoistNotInCalibrationZone" : Bool = PLC HMI_DB.Calibration.Trolley.PrerequisitesNotOK AT %DB1.DBX0.0, 1 s
   "HMI_DB_Calibration_Trolley_CurrentStep" : UInt = PLC HMI_DB.Calibration.Trolley.CurrentStep AT %DB1.DBX0.0, 1 s
   "HMI_DB_Calibration_Trolley_CompletedSteps" : DWord = PLC HMI_DB.Calibration.Trolley.CompletedSteps AT %DB1.DBX0.0, 1 s
   "HMI_DB_Calibration_Trolley_Reference3K1" : Bool = PLC HMI_DB.Calibration.Trolley.Reference3K1 AT %DB1.DBX0.0, 1 s
   "HMI_DB_Calibration_Trolley_Position_mm" : DInt = PLC HMI_DB.Calibration.Trolley.Position_mm AT %DB1.DBX0.0, 1 s
   "HMI_DB_Calibration_Trolley_DriveVelocity_rpm" : Real = PLC HMI_DB.Calibration.Trolley.DriveVelocity_rpm AT %DB1.DBX0.0, 1 s
   "HMI_DB_Calibration_Trolley_TimerRemaining" : Time = PLC HMI_DB.Calibration.Trolley.TimerRemaining AT %DB1.DBX0.0, 1 s
   "HMI_DB_Calibration_Trolley_TimerRemaining_Min" : UInt = PLC HMI_DB.Calibration.Trolley.TimerRemaining_Min AT %DB1.DBX0.0, 1 s
   "HMI_DB_Calibration_Trolley_TimerRemaining_Sec" : UInt = PLC HMI_DB.Calibration.Trolley.TimerRemaining_Sec AT %DB1.DBX0.0, 1 s
   "HMI_DB_Calibration_Trolley_Steps_Completed_Step10" : Bool = PLC HMI_DB.Calibration.Trolley.Steps_Completed.Step10 AT %DB1.DBX0.0, 1 s
   "HMI_DB_Calibration_Trolley_Steps_Completed_Step20" : Bool = PLC HMI_DB.Calibration.Trolley.Steps_Completed.Step20 AT %DB1.DBX0.0, 1 s
   "HMI_DB_Calibration_Trolley_Steps_Completed_Step30" : Bool = PLC HMI_DB.Calibration.Trolley.Steps_Completed.Step30 AT %DB1.DBX0.0, 1 s
   "HMI_DB_Calibration_Trolley_Steps_Completed_Step40" : Bool = PLC HMI_DB.Calibration.Trolley.Steps_Completed.Step40 AT %DB1.DBX0.0, 1 s
   "HMI_DB_Calibration_Trolley_Steps_Completed_Step50" : Bool = PLC HMI_DB.Calibration.Trolley.Steps_Completed.Step50 AT %DB1.DBX0.0, 1 s
   "HMI_DB_Calibration_Trolley_Steps_Completed_Step60" : Bool = PLC HMI_DB.Calibration.Trolley.Steps_Completed.Step60 AT %DB1.DBX0.0, 1 s
   "HMI_DB_Calibration_Trolley_Steps_Completed_Step70" : Bool = PLC HMI_DB.Calibration.Trolley.Steps_Completed.Step70 AT %DB1.DBX0.0, 1 s
   "HMI_DB_Calibration_Trolley_Steps_Completed_Step80" : Bool = PLC HMI_DB.Calibration.Trolley.Steps_Completed.Step80 AT %DB1.DBX0.0, 1 s
   "HMI_DB_Calibration_Trolley_Steps_Completed_Step90" : Bool = PLC HMI_DB.Calibration.Trolley.Steps_Completed.Step90 AT %DB1.DBX0.0, 1 s
   "HMI_DB_Calibration_Trolley_Steps_Completed_Step100" : Bool = PLC HMI_DB.Calibration.Trolley.Steps_Completed.Step100 AT %DB1.DBX0.0, 1 s
   "HMI_DB_Calibration_Trolley_Steps_Completed_Step110" : Bool = PLC HMI_DB.Calibration.Trolley.Steps_Completed.Step110 AT %DB1.DBX0.0, 1 s
   "HMI_DB_Calibration_Trolley_Steps_Completed_Step120" : Bool = PLC HMI_DB.Calibration.Trolley.Steps_Completed.Step120 AT %DB1.DBX0.0, 1 s
   "HMI_DB_Calibration_Trolley_Steps_Completed_Step130" : Bool = PLC HMI_DB.Calibration.Trolley.Steps_Completed.Step130 AT %DB1.DBX0.0, 1 s
   "HMI_DB_Calibration_Trolley_Steps_Active_Step10" : Bool = PLC HMI_DB.Calibration.Trolley.Steps_Active.Step10 AT %DB1.DBX0.0, 1 s
   "HMI_DB_Calibration_Trolley_Steps_Active_Step20" : Bool = PLC HMI_DB.Calibration.Trolley.Steps_Active.Step20 AT %DB1.DBX0.0, 1 s
   "HMI_DB_Calibration_Trolley_Steps_Active_Step30" : Bool = PLC HMI_DB.Calibration.Trolley.Steps_Active.Step30 AT %DB1.DBX0.0, 1 s
   "HMI_DB_Calibration_Trolley_Steps_Active_Step40" : Bool = PLC HMI_DB.Calibration.Trolley.Steps_Active.Step40 AT %DB1.DBX0.0, 1 s
   "HMI_DB_Calibration_Trolley_Steps_Active_Step50" : Bool = PLC HMI_DB.Calibration.Trolley.Steps_Active.Step50 AT %DB1.DBX0.0, 1 s
   "HMI_DB_Calibration_Trolley_Steps_Active_Step60" : Bool = PLC HMI_DB.Calibration.Trolley.Steps_Active.Step60 AT %DB1.DBX0.0, 1 s
   "HMI_DB_Calibration_Trolley_Steps_Active_Step70" : Bool = PLC HMI_DB.Calibration.Trolley.Steps_Active.Step70 AT %DB1.DBX0.0, 1 s
   "HMI_DB_Calibration_Trolley_Steps_Active_Step80" : Bool = PLC HMI_DB.Calibration.Trolley.Steps_Active.Step80 AT %DB1.DBX0.0, 1 s
   "HMI_DB_Calibration_Trolley_Steps_Active_Step90" : Bool = PLC HMI_DB.Calibration.Trolley.Steps_Active.Step90 AT %DB1.DBX0.0, 1 s
   "HMI_DB_Calibration_Trolley_Steps_Active_Step100" : Bool = PLC HMI_DB.Calibration.Trolley.Steps_Active.Step100 AT %DB1.DBX0.0, 1 s
   "HMI_DB_Calibration_Trolley_Steps_Active_Step110" : Bool = PLC HMI_DB.Calibration.Trolley.Steps_Active.Step110 AT %DB1.DBX0.0, 1 s
   "HMI_DB_Calibration_Trolley_Steps_Active_Step120" : Bool = PLC HMI_DB.Calibration.Trolley.Steps_Active.Step120 AT %DB1.DBX0.0, 1 s
   "HMI_DB_Calibration_Trolley_Steps_Active_Step130" : Bool = PLC HMI_DB.Calibration.Trolley.Steps_Active.Step130 AT %DB1.DBX0.0, 1 s
   "HMI_DB_Calibration_Trolley_Diagnostics_EncoderControlHealthy" : Bool = PLC HMI_DB.Calibration.Trolley.Diagnostics.EncoderControlHealthy AT %DB1.DBX0.0, 1 s
   "HMI_DB_Calibration_Trolley_Diagnostics_StartupDataConsistent" : Bool = PLC HMI_DB.Calibration.Trolley.Diagnostics.StartupDataConsistent AT %DB1.DBX0.0, 1 s
   "HMI_DB_Calibration_Trolley_Diagnostics_NoMovementWithoutCommand" : Bool = PLC HMI_DB.Calibration.Trolley.Diagnostics.NoMovementWithoutCommand AT %DB1.DBX0.0, 1 s
   "HMI_DB_Calibration_Trolley_Diagnostics_NoManualMovementDetected" : Bool = PLC HMI_DB.Calibration.Trolley.Diagnostics.NoManualMovementDetected AT %DB1.DBX0.0, 1 s
   "HMI_DB_Calibration_Trolley_Diagnostics_EncoderUpdatesDuringMotion" : Bool = PLC HMI_DB.Calibration.Trolley.Diagnostics.EncoderUpdatesDuringMotion AT %DB1.DBX0.0, 1 s
   "HMI_DB_Calibration_Trolley_Diagnostics_EncoderReplacementNotDetected" : Bool = PLC HMI_DB.Calibration.Trolley.Diagnostics.EncoderReplacementNotDetected AT %DB1.DBX0.0, 1 s
   "HMI_DB_Calibration_Trolley_PrerequisitesNotOK" : Bool = PLC HMI_DB.Calibration.Trolley.PrerequisitesNotOK AT %DB1.DBX0.0, 1 s

HMI tags "CraneMovementMechanism"
   "HMI_DB_Crane_movement_mechanism_Brake_protection_On" : Bool = PLC HMI_DB.Crane_movement_mechanism.Brake_protection_On, 1 s
   "HMI_DB_Crane_movement_mechanism_4M1_engine_temperature_protection" : Bool = PLC HMI_DB.Crane_movement_mechanism.4M1_engine_temperature_protection, 1 s
   "HMI_DB_Crane_movement_mechanism_4M2_engine_temperature_protection" : Bool = PLC HMI_DB.Crane_movement_mechanism.4M2_engine_temperature_protection, 1 s
   "HMI_DB_Crane_movement_mechanism_WP_Either_side_column" : Bool = PLC HMI_DB.Crane_movement_mechanism.WP_Either_side_column, 1 s
   "HMI_DB_Crane_movement_mechanism_4RT1_thermal_protection_braking_resistor" : Bool = PLC HMI_DB.Crane_movement_mechanism.4RT1_thermal_protection_braking_resistor, 1 s
   "HMI_DB_Crane_movement_mechanism_4RT2_thermal_protection_braking_resistor" : Bool = PLC HMI_DB.Crane_movement_mechanism.4RT2_thermal_protection_braking_resistor, 1 s
   "HMI_DB_Crane_movement_mechanism_NSP_Left_movement" : Bool = PLC HMI_DB.Crane_movement_mechanism.NSP_Left_movement, 1 s
   "HMI_DB_Crane_movement_mechanism_NSP_Right_movement" : Bool = PLC HMI_DB.Crane_movement_mechanism.NSP_Right_movement, 1 s
   "HMI_DB_Crane_movement_mechanism_WP_Left_movement" : Bool = PLC HMI_DB.Crane_movement_mechanism.WP_Left_movement, 1 s
   "HMI_DB_Crane_movement_mechanism_WP_Right_movement" : Bool = PLC HMI_DB.Crane_movement_mechanism.WP_Right_movement, 1 s
   "HMI_DB_Crane_movement_mechanism_4SQ41_MD_disconnected_from_drive" : Bool = PLC HMI_DB.Crane_movement_mechanism.4SQ41_MD_disconnected_from_drive, 1 s
   "HMI_DB_Crane_movement_mechanism_4SQ42_MD_disconnected_from_drive" : Bool = PLC HMI_DB.Crane_movement_mechanism.4SQ42_MD_disconnected_from_drive, 1 s
   "HMI_DB_Crane_movement_mechanism_CMD_Service_brake_On" : Bool = PLC HMI_DB.Crane_movement_mechanism.CMD_Service_brake_On, 1 s
   "HMI_DB_Crane_movement_mechanism_HL_Drive_ready" : Bool = PLC HMI_DB.Crane_movement_mechanism.HL_Drive_ready, 1 s
   "HMI_DB_Crane_movement_mechanism_NSP_Enable_movement" : Bool = PLC HMI_DB.Crane_movement_mechanism.NSP_Enable_movement AT %DB1.DBX0.0, 1 s
   "HMI_DB_Crane_movement_mechanism_BreakThermalProtection" : Bool = PLC HMI_DB.Crane_movement_mechanism.BreakThermalProtection AT %DB1.DBX0.0, 1 s
   "HMI_DB_Crane_movement_mechanism_MotorThermalProtection" : Bool = PLC HMI_DB.Crane_movement_mechanism.MotorThermalProtection AT %DB1.DBX0.0, 1 s
   "HMI_DB_Crane_movement_mechanism_SecondSpeedLeft" : Bool = PLC HMI_DB.Crane_movement_mechanism.SecondSpeedLeft AT %DB1.DBX0.0, 1 s
   "HMI_DB_Crane_movement_mechanism_SecondSpeedRight" : Bool = PLC HMI_DB.Crane_movement_mechanism.SecondSpeedRight AT %DB1.DBX0.0, 1 s
   "HMI_DB_Crane_movement_mechanism_FirstSpeedLeft" : Bool = PLC HMI_DB.Crane_movement_mechanism.FirstSpeedLeft AT %DB1.DBX0.0, 1 s
   "HMI_DB_Crane_movement_mechanism_FirstSpeedRight" : Bool = PLC HMI_DB.Crane_movement_mechanism.FirstSpeedRight AT %DB1.DBX0.0, 1 s
   "HMI_DB_Crane_movement_mechanism_CM_Status" : Word = PLC HMI_DB.Crane_movement_mechanism.CM_Status AT %DB1.DBX0.0, 1 s
   "HMI_DB_Calibration_Crane_Active" : Bool = PLC HMI_DB.Calibration.Crane.Active AT %DB1.DBX0.0, 1 s
   "HMI_DB_Calibration_Crane_Calibrated" : Bool = PLC HMI_DB.Calibration.Crane.Calibrated AT %DB1.DBX0.0, 1 s
   "HMI_DB_Calibration_Crane_Fault" : Bool = PLC HMI_DB.Calibration.Crane.Fault AT %DB1.DBX0.0, 1 s
   "HMI_DB_Calibration_Crane_Aborted" : Bool = PLC HMI_DB.Calibration.Crane.Aborted AT %DB1.DBX0.0, 1 s
   "HMI_DB_Calibration_Crane_PrerequisitesNotOK" : Bool = PLC HMI_DB.Calibration.Crane.PrerequisitesNotOK AT %DB1.DBX0.0, 1 s
   "HMI_DB_Calibration_Crane_CurrentStep" : UInt = PLC HMI_DB.Calibration.Crane.CurrentStep AT %DB1.DBX0.0, 1 s
   "HMI_DB_Calibration_Crane_CompletedSteps" : DWord = PLC HMI_DB.Calibration.Crane.CompletedSteps AT %DB1.DBX0.0, 1 s
   "HMI_DB_Calibration_Crane_Reference4K1" : Bool = PLC HMI_DB.Calibration.Crane.Reference4K1 AT %DB1.DBX0.0, 1 s
   "HMI_DB_Calibration_Crane_Position4BR1_mm" : DInt = PLC HMI_DB.Calibration.Crane.Position4BR1_mm AT %DB1.DBX0.0, 1 s
   "HMI_DB_Calibration_Crane_Position4BR2_mm" : DInt = PLC HMI_DB.Calibration.Crane.Position4BR2_mm AT %DB1.DBX0.0, 1 s
   "HMI_DB_Calibration_Crane_Drive1Velocity_rpm" : Real = PLC HMI_DB.Calibration.Crane.Drive1Velocity_rpm AT %DB1.DBX0.0, 1 s
   "HMI_DB_Calibration_Crane_Drive2Velocity_rpm" : Real = PLC HMI_DB.Calibration.Crane.Drive2Velocity_rpm AT %DB1.DBX0.0, 1 s
   "HMI_DB_Calibration_Crane_TimerRemaining" : Time = PLC HMI_DB.Calibration.Crane.TimerRemaining AT %DB1.DBX0.0, 1 s
   "HMI_DB_Calibration_Crane_TimerRemaining_Min" : UInt = PLC HMI_DB.Calibration.Crane.TimerRemaining_Min AT %DB1.DBX0.0, 1 s
   "HMI_DB_Calibration_Crane_TimerRemaining_Sec" : UInt = PLC HMI_DB.Calibration.Crane.TimerRemaining_Sec AT %DB1.DBX0.0, 1 s
   "HMI_DB_Calibration_Crane_Steps_Completed_Step10" : Bool = PLC HMI_DB.Calibration.Crane.Steps_Completed.Step10 AT %DB1.DBX0.0, 1 s
   "HMI_DB_Calibration_Crane_Steps_Completed_Step20" : Bool = PLC HMI_DB.Calibration.Crane.Steps_Completed.Step20 AT %DB1.DBX0.0, 1 s
   "HMI_DB_Calibration_Crane_Steps_Completed_Step30" : Bool = PLC HMI_DB.Calibration.Crane.Steps_Completed.Step30 AT %DB1.DBX0.0, 1 s
   "HMI_DB_Calibration_Crane_Steps_Completed_Step40" : Bool = PLC HMI_DB.Calibration.Crane.Steps_Completed.Step40 AT %DB1.DBX0.0, 1 s
   "HMI_DB_Calibration_Crane_Steps_Completed_Step50" : Bool = PLC HMI_DB.Calibration.Crane.Steps_Completed.Step50 AT %DB1.DBX0.0, 1 s
   "HMI_DB_Calibration_Crane_Steps_Completed_Step60" : Bool = PLC HMI_DB.Calibration.Crane.Steps_Completed.Step60 AT %DB1.DBX0.0, 1 s
   "HMI_DB_Calibration_Crane_Steps_Completed_Step70" : Bool = PLC HMI_DB.Calibration.Crane.Steps_Completed.Step70 AT %DB1.DBX0.0, 1 s
   "HMI_DB_Calibration_Crane_Steps_Completed_Step80" : Bool = PLC HMI_DB.Calibration.Crane.Steps_Completed.Step80 AT %DB1.DBX0.0, 1 s
   "HMI_DB_Calibration_Crane_Steps_Completed_Step90" : Bool = PLC HMI_DB.Calibration.Crane.Steps_Completed.Step90 AT %DB1.DBX0.0, 1 s
   "HMI_DB_Calibration_Crane_Steps_Completed_Step100" : Bool = PLC HMI_DB.Calibration.Crane.Steps_Completed.Step100 AT %DB1.DBX0.0, 1 s
   "HMI_DB_Calibration_Crane_Steps_Completed_Step110" : Bool = PLC HMI_DB.Calibration.Crane.Steps_Completed.Step110 AT %DB1.DBX0.0, 1 s
   "HMI_DB_Calibration_Crane_Steps_Completed_Step120" : Bool = PLC HMI_DB.Calibration.Crane.Steps_Completed.Step120 AT %DB1.DBX0.0, 1 s
   "HMI_DB_Calibration_Crane_Steps_Completed_Step130" : Bool = PLC HMI_DB.Calibration.Crane.Steps_Completed.Step130 AT %DB1.DBX0.0, 1 s
   "HMI_DB_Calibration_Crane_Steps_Active_Step10" : Bool = PLC HMI_DB.Calibration.Crane.Steps_Active.Step10 AT %DB1.DBX0.0, 1 s
   "HMI_DB_Calibration_Crane_Steps_Active_Step20" : Bool = PLC HMI_DB.Calibration.Crane.Steps_Active.Step20 AT %DB1.DBX0.0, 1 s
   "HMI_DB_Calibration_Crane_Steps_Active_Step30" : Bool = PLC HMI_DB.Calibration.Crane.Steps_Active.Step30 AT %DB1.DBX0.0, 1 s
   "HMI_DB_Calibration_Crane_Steps_Active_Step40" : Bool = PLC HMI_DB.Calibration.Crane.Steps_Active.Step40 AT %DB1.DBX0.0, 1 s
   "HMI_DB_Calibration_Crane_Steps_Active_Step50" : Bool = PLC HMI_DB.Calibration.Crane.Steps_Active.Step50 AT %DB1.DBX0.0, 1 s
   "HMI_DB_Calibration_Crane_Steps_Active_Step60" : Bool = PLC HMI_DB.Calibration.Crane.Steps_Active.Step60 AT %DB1.DBX0.0, 1 s
   "HMI_DB_Calibration_Crane_Steps_Active_Step70" : Bool = PLC HMI_DB.Calibration.Crane.Steps_Active.Step70 AT %DB1.DBX0.0, 1 s
   "HMI_DB_Calibration_Crane_Steps_Active_Step80" : Bool = PLC HMI_DB.Calibration.Crane.Steps_Active.Step80 AT %DB1.DBX0.0, 1 s
   "HMI_DB_Calibration_Crane_Steps_Active_Step90" : Bool = PLC HMI_DB.Calibration.Crane.Steps_Active.Step90 AT %DB1.DBX0.0, 1 s
   "HMI_DB_Calibration_Crane_Steps_Active_Step100" : Bool = PLC HMI_DB.Calibration.Crane.Steps_Active.Step100 AT %DB1.DBX0.0, 1 s
   "HMI_DB_Calibration_Crane_Steps_Active_Step110" : Bool = PLC HMI_DB.Calibration.Crane.Steps_Active.Step110 AT %DB1.DBX0.0, 1 s
   "HMI_DB_Calibration_Crane_Steps_Active_Step120" : Bool = PLC HMI_DB.Calibration.Crane.Steps_Active.Step120 AT %DB1.DBX0.0, 1 s
   "HMI_DB_Calibration_Crane_Steps_Active_Step130" : Bool = PLC HMI_DB.Calibration.Crane.Steps_Active.Step130 AT %DB1.DBX0.0, 1 s
   "HMI_DB_Calibration_Crane_Diagnostics_Encoder1ControlHealthy" : Bool = PLC HMI_DB.Calibration.Crane.Diagnostics.Encoder1ControlHealthy AT %DB1.DBX0.0, 1 s
   "HMI_DB_Calibration_Crane_Diagnostics_Encoder1StartupDataConsistent" : Bool = PLC HMI_DB.Calibration.Crane.Diagnostics.Encoder1StartupDataConsistent AT %DB1.DBX0.0, 1 s
   "HMI_DB_Calibration_Crane_Diagnostics_Encoder1NoMovementWithoutCommand" : Bool = PLC HMI_DB.Calibration.Crane.Diagnostics.Encoder1NoMovementWithoutCommand AT %DB1.DBX0.0, 1 s
   "HMI_DB_Calibration_Crane_Diagnostics_Encoder1NoManualMovementDetected" : Bool = PLC HMI_DB.Calibration.Crane.Diagnostics.Encoder1NoManualMovementDetected AT %DB1.DBX0.0, 1 s
   "HMI_DB_Calibration_Crane_Diagnostics_Encoder1UpdatesDuringMotion" : Bool = PLC HMI_DB.Calibration.Crane.Diagnostics.Encoder1UpdatesDuringMotion AT %DB1.DBX0.0, 1 s
   "HMI_DB_Calibration_Crane_Diagnostics_Encoder1ReplacementNotDetected" : Bool = PLC HMI_DB.Calibration.Crane.Diagnostics.Encoder1ReplacementNotDetected AT %DB1.DBX0.0, 1 s
   "HMI_DB_Calibration_Crane_Diagnostics_Encoder2ControlHealthy" : Bool = PLC HMI_DB.Calibration.Crane.Diagnostics.Encoder2ControlHealthy AT %DB1.DBX0.0, 1 s
   "HMI_DB_Calibration_Crane_Diagnostics_Encoder2StartupDataConsistent" : Bool = PLC HMI_DB.Calibration.Crane.Diagnostics.Encoder2StartupDataConsistent AT %DB1.DBX0.0, 1 s
   "HMI_DB_Calibration_Crane_Diagnostics_Encoder2NoMovementWithoutCommand" : Bool = PLC HMI_DB.Calibration.Crane.Diagnostics.Encoder2NoMovementWithoutCommand AT %DB1.DBX0.0, 1 s
   "HMI_DB_Calibration_Crane_Diagnostics_Encoder2NoManualMovementDetected" : Bool = PLC HMI_DB.Calibration.Crane.Diagnostics.Encoder2NoManualMovementDetected AT %DB1.DBX0.0, 1 s
   "HMI_DB_Calibration_Crane_Diagnostics_Encoder2UpdatesDuringMotion" : Bool = PLC HMI_DB.Calibration.Crane.Diagnostics.Encoder2UpdatesDuringMotion AT %DB1.DBX0.0, 1 s
   "HMI_DB_Calibration_Crane_Diagnostics_Encoder2ReplacementNotDetected" : Bool = PLC HMI_DB.Calibration.Crane.Diagnostics.Encoder2ReplacementNotDetected AT %DB1.DBX0.0, 1 s
   "HMI_DB_Calibration_Crane_Diagnostics_EncoderDifferenceOK" : Bool = PLC HMI_DB.Calibration.Crane.Diagnostics.EncoderDifferenceOK AT %DB1.DBX0.0, 1 s
   "HMI_DB_Calibration_Crane_Diagnostics_DiagnosticsHealthy" : Bool = PLC HMI_DB.Calibration.Crane.Diagnostics.DiagnosticsHealthy AT %DB1.DBX0.0, 1 s
   "HMI_DB_Calibration_Crane_Diagnostics_DriveStandstill" : Bool = PLC HMI_DB.Calibration.Crane.Diagnostics.DriveStandstill AT %DB1.DBX0.0, 1 s
   "HMI_DB_Calibration_Crane_Diagnostics_EncoderDifference_mm" : LReal = PLC HMI_DB.Calibration.Crane.Diagnostics.EncoderDifference_mm AT %DB1.DBX0.0, 1 s
   "HMI_DB_Calibration_Crane_Diagnostics_Position1DeltaStopped_mm" : LReal = PLC HMI_DB.Calibration.Crane.Diagnostics.Position1DeltaStopped_mm AT %DB1.DBX0.0, 1 s
   "HMI_DB_Calibration_Crane_Diagnostics_Position2DeltaStopped_mm" : LReal = PLC HMI_DB.Calibration.Crane.Diagnostics.Position2DeltaStopped_mm AT %DB1.DBX0.0, 1 s
   "HMI_DB_Calibration_Crane_Diagnostics_Position1DeltaMotion_mm" : LReal = PLC HMI_DB.Calibration.Crane.Diagnostics.Position1DeltaMotion_mm AT %DB1.DBX0.0, 1 s
   "HMI_DB_Calibration_Crane_Diagnostics_Position2DeltaMotion_mm" : LReal = PLC HMI_DB.Calibration.Crane.Diagnostics.Position2DeltaMotion_mm AT %DB1.DBX0.0, 1 s

HMI tags "MessagesContactor"
   "HMI_DB_Messages_LinearContactor_wMessageWord1" : Word = PLC HMI_DB.Messages.LinearContactor.wMessageWord1, 1 s
   "HMI_DB_Messages_LinearContactor_wMessageWord2" : Word = PLC HMI_DB.Messages.LinearContactor.wMessageWord2, 1 s
   "HMI_DB_Messages_LinearContactor_wMessageWord3" : Word = PLC HMI_DB.Messages.LinearContactor.wMessageWord3, 1 s
   "HMI_DB_Messages_LinearContactor_wMessageWord4" : Word = PLC HMI_DB.Messages.LinearContactor.wMessageWord4, 1 s
   "HMI_DB_Messages_LinearContactor_wMessageWord5" : Word = PLC HMI_DB.Messages.LinearContactor.wMessageWord5, 1 s

HMI tags "ButtonHighlight"
   "HMI_DB_wButtonHighlight" : Word = PLC HMI_DB.wButtonHighlight, 1 s

HMI tags "Drives"
   "HMI_DB_Drives_CU_U1" : UDT_HMI_S120_CU = PLC HMI_DB.Drives.CU_U1, 1 s
   "HMI_DB_Drives_Drive_1UZ1" : UDT_HMI_S120_Drive = PLC HMI_DB.Drives.Drive_1UZ1 AT %DB1.DBW0, 1 s
   "HMI_DB_Drives_Drive_3UZ1" : UDT_HMI_S120_Drive = PLC HMI_DB.Drives.Drive_3UZ1 AT %DB1.DBW0, 1 s
   "HMI_DB_Drives_Drive_4UZ1" : UDT_HMI_S120_Drive = PLC HMI_DB.Drives.Drive_4UZ1 AT %DB1.DBW0, 1 s
   "HMI_DB_Drives_Drive_4UZ2" : UDT_HMI_S120_Drive = PLC HMI_DB.Drives.Drive_4UZ2 AT %DB1.DBW0, 1 s

HMI tags "MessagesLiftUp"
   "HMI_DB_Messages_LiftUp_wMessageWord1" : Word = PLC HMI_DB.Messages.LiftUp.wMessageWord1, 1 s
   "HMI_DB_Messages_LiftUp_wMessageWord2" : Word = PLC HMI_DB.Messages.LiftUp.wMessageWord2, 1 s
   "HMI_DB_Messages_LiftUp_wMessageWord3" : Word = PLC HMI_DB.Messages.LiftUp.wMessageWord3, 1 s
   "HMI_DB_Messages_LiftUp_wMessageWord4" : Word = PLC HMI_DB.Messages.LiftUp.wMessageWord4 AT %DB1.DBW0, 1 s

HMI tags "Diagnostics"
   "HMI_DB_Messages_Diag_wMessageWord1" : Word = PLC HMI_DB.Messages.Diag.wMessageWord1, 1 s
   "HMI_DB_Messages_Diag_wMessageWord2" : Word = PLC HMI_DB.Messages.Diag.wMessageWord2 AT %DB1.DBW0, 1 s

HMI tags "LiftUpErrors"
   "HMI_DB_Alarms_LiftUp_AlarmWord1" : Word = PLC HMI_DB.Alarms.LiftUp.AlarmWord1, 1 s
   "HMI_DB_Alarms_LiftUp_AlarmWord2" : Word = PLC HMI_DB.Alarms.LiftUp.AlarmWord2 AT %DB1.DBW0, 1 s
   "HMI_DB_Warnings_LiftUp" : Word = PLC HMI_DB.Warnings.LiftUp AT %DB1.DBW0, 1 s

HMI tags "MessagesTrolley"
   "HMI_DB_Messages_Trolley_wMessageWord1" : Word = PLC HMI_DB.Messages.Trolley.wMessageWord1, 1 s
   "HMI_DB_Messages_Trolley_wMessageWord2" : Word = PLC HMI_DB.Messages.Trolley.wMessageWord2, 1 s
   "HMI_DB_Messages_Trolley_wMessageWord3" : Word = PLC HMI_DB.Messages.Trolley.wMessageWord3, 1 s

HMI tags "TrolleyMovementErrors"
   "HMI_DB_Alarms_Trolley_AlarmWord1" : Word = PLC HMI_DB.Alarms.Trolley.AlarmWord1, 1 s
   "HMI_DB_Alarms_Trolley_AlarmWord2" : Word = PLC HMI_DB.Alarms.Trolley.AlarmWord2 AT %DB1.DBW0, 1 s
   "HMI_DB_Warnings_Trolley" : Word = PLC HMI_DB.Warnings.Trolley AT %DB1.DBW0, 1 s

HMI tags "MessagesCrane"
   "HMI_DB_Messages_Crane_wMessageWord3" : Word = PLC HMI_DB.Messages.Crane.wMessageWord3, 1 s
   "HMI_DB_Messages_Crane_wMessageWord2" : Word = PLC HMI_DB.Messages.Crane.wMessageWord2 AT %DB1.DBW0, 1 s
   "HMI_DB_Messages_Crane_wMessageWord1" : Word = PLC HMI_DB.Messages.Crane.wMessageWord1 AT %DB1.DBW0, 1 s

HMI tags "CraneErrors"
   "HMI_DB_Alarms_Crane_AlarmWord1" : Word = PLC HMI_DB.Alarms.Crane.AlarmWord1, 1 s
   "HMI_DB_Alarms_Crane_AlarmWord2" : Word = PLC HMI_DB.Alarms.Crane.AlarmWord2 AT %DB1.DBW0, 1 s
   "HMI_DB_Warnings_Crane" : Word = PLC HMI_DB.Warnings.Crane AT %DB1.DBW0, 1 s

HMI tags "Self"
   "HMI_DB_Messages_Self_wMessageWord1" : Word = PLC HMI_DB.Messages.Self.wMessageWord1, 1 s

HMI tags "Diagnose"
   "HMI_DB_Alarms_Diagn_AlarmWord1" : Word = PLC HMI_DB.Alarms.Diagnose.AlarmWord1 AT %DB1.DBW0, 1 s
   "Lifebit_HMI" : Bool = PLC Data_base.Lifebit_HMI AT %DB1.DBX22.1, 1 s
   "HMI_DB_Diagnostics_Ring_PLC_HMI_NOK" : Bool = PLC HMI_DB.Diagnostics.Ring_PLC_HMI_NOK AT %DB1.DBW0, 1 s
      on ChangeValue: "HMI_UpdateCommunication"()
   "HMI_DB_Diagnostics_Ring_PLC_SCALAMCE_NOK" : Bool = PLC HMI_DB.Diagnostics.Ring_PLC_SCALAMCE_NOK AT %DB1.DBW0, 1 s
      on ChangeValue: "HMI_UpdateCommunication"()
   "HMI_DB_Diagnostics_Ring_HMI_CU_NOK" : Bool = PLC HMI_DB.Diagnostics.Ring_HMI_CU_NOK AT %DB1.DBW0, 1 s
      on ChangeValue: "HMI_UpdateCommunication"()
   "HMI_DB_Diagnostics_Ring_SCALAMCE_CU_NOK" : Bool = PLC HMI_DB.Diagnostics.Ring_SCALAMCE_CU_NOK AT %DB1.DBW0, 1 s
      on ChangeValue: "HMI_UpdateCommunication"()
   "PLC_Clock_1Hz" : Bool = PLC Clock_1Hz AT %M0.5, 100 ms
      on ChangeValue: InvertBit("Lifebit_HMI")
   "PN_Diagnostics_DisplayOpen" : Bool = PLC DB_Diag_Prof.DisplayOpen AT %DB1.DBW0, 1 s
      on ChangeValue: "HMI_UpdateCommunication"()
   "PN_Diagnostics_DisplayClosed" : Bool = PLC DB_Diag_Prof.DisplayClosed AT %DB1.DBW0, 1 s
      on ChangeValue: "HMI_UpdateCommunication"()
   "PN_Diagnostics_DisplayUnknown" : Bool = PLC DB_Diag_Prof.DisplayUnknown AT %DB1.DBW0, 1 s
      on ChangeValue: "HMI_UpdateCommunication"()
   "PN_Diagnostics_DisplayHmiFault" : Bool = PLC DB_Diag_Prof.DisplayHmiNoFault AT %DB1.DBW0, 1 s
      on ChangeValue: "HMI_UpdateCommunication"()
   "HMI_PLC_Available" : Bool = PLC DB_HMI_Connection.Available AT %DB631.DBX0.0, 100 ms   // Резервний старий тег. Не використовується для визначення стану звʼязку або видимості повідомлень.
   "HMI_Coordination" : Word = PLC HMI_DB.wCoordination AT %DB1.DBW0, 100 ms   // Існуюче слово області Coordination: HMI_DB.wCoordination. Панель змінює контрольний біт навіть у STOP ПЛК. Подія зміни опитує режим ПЛК.
      on ChangeValue: function_c655a98f("HMI_Connection_1", "HMI_PLC_Mode"); "HMI_UpdateCommunication"()
   "HMI_PLC_Mode" : Int, internal   // Локальний результат GetPLCMode: 4 — STOP, 8 — RUN, 0 — ще не визначено. Не зберігається у ПЛК.
      on ChangeValue: "HMI_UpdateCommunication"()
   "HMI_Show_NoConnection" : Bool, internal   // Внутрішній стан зʼєднання HMI. Системна подія 140001 встановлює 1, 140000 встановлює 0. Початково 1. Не визначається за кешованими тегами ПЛК.
      on ChangeValue: "HMI_UpdateCommunication"()
   "HMI_Show_CpuStopped" : Bool, internal   // Локальна ознака індикації. Обчислюється скриптом HMI_UpdateCommunication з урахуванням доступності ПЛК та режиму RUN.
   "HMI_Show_CpuUnknown" : Bool, internal   // Локальна ознака індикації. Обчислюється скриптом HMI_UpdateCommunication з урахуванням доступності ПЛК та режиму RUN.
   "HMI_Show_RingOpen" : Bool, internal   // Локальна ознака індикації. Обчислюється скриптом HMI_UpdateCommunication з урахуванням доступності ПЛК та режиму RUN.
   "HMI_Show_RingClosed" : Bool, internal   // Локальна ознака індикації. Обчислюється скриптом HMI_UpdateCommunication з урахуванням доступності ПЛК та режиму RUN.
   "HMI_Show_DiagnosticsUnknown" : Bool, internal   // Локальна ознака індикації. Обчислюється скриптом HMI_UpdateCommunication з урахуванням доступності ПЛК та режиму RUN.
   "HMI_Show_PanelFault" : Bool, internal   // Локальна ознака індикації. Обчислюється скриптом HMI_UpdateCommunication з урахуванням доступності ПЛК та режиму RUN.
   "HMI_Show_Cross_PLC_HMI" : Bool, internal   // Локальна ознака індикації. Обчислюється скриптом HMI_UpdateCommunication з урахуванням доступності ПЛК та режиму RUN.
   "HMI_Show_Cross_PLC_SC" : Bool, internal   // Локальна ознака індикації. Обчислюється скриптом HMI_UpdateCommunication з урахуванням доступності ПЛК та режиму RUN.
   "HMI_Show_Cross_SC_CU" : Bool, internal   // Локальна ознака індикації. Обчислюється скриптом HMI_UpdateCommunication з урахуванням доступності ПЛК та режиму RUN.
   "HMI_Show_Cross_HMI_CU" : Bool, internal   // Локальна ознака індикації. Обчислюється скриптом HMI_UpdateCommunication з урахуванням доступності ПЛК та режиму RUN.

